Staubli VAL3: XHS3023L2.dtx

public frame fPartReal = {x=0.000, y=0.000, z=0.000, rx=0.000, ry=0.000, rz=0.000, fatherId=world[0]}
public jointRx jtPark = {j1=-10.678, j2=62.119, j3=50.568, j4=-4.773, j5=72.927, j6=-11.595}
public jointRx ptRoutingPath[1367]
  [0] = {j1=-10.951, j2=61.954, j3=48.631, j4=-3.846, j5=78.024, j6=-9.408}
  [1] = {j1=-10.927, j2=62.459, j3=48.172, j4=-3.903, j5=78.392, j6=-8.968}
  [2] = {j1=-10.905, j2=62.967, j3=47.706, j4=-3.960, j5=78.777, j6=-8.517}
  [3] = {j1=-10.884, j2=63.472, j3=47.245, j4=-4.014, j5=79.163, j6=-8.066}
  [4] = {j1=-10.866, j2=63.967, j3=46.802, j4=-4.064, j5=79.533, j6=-7.626}
  [5] = {j1=-10.851, j2=64.445, j3=46.388, j4=-4.105, j5=79.872, j6=-7.209}
  [6] = {j1=-10.848, j2=64.525, j3=46.320, j4=-4.112, j5=79.926, j6=-7.139}
  [7] = {j1=-10.829, j2=64.971, j3=45.959, j4=-4.174, j5=80.205, j6=-6.748}
  [8] = {j1=-10.797, j2=65.452, j3=45.616, j4=-4.291, j5=80.435, j6=-6.319}
  [9] = {j1=-10.755, j2=65.869, j3=45.388, j4=-4.456, j5=80.522, j6=-5.949}
  [10] = {j1=-10.719, j2=66.156, j3=45.303, j4=-4.610, j5=80.466, j6=-5.711}
  [11] = {j1=-10.683, j2=66.396, j3=45.302, j4=-4.767, j5=80.303, j6=-5.536}
  [12] = {j1=-10.648, j2=66.596, j3=45.373, j4=-4.931, j5=80.045, j6=-5.415}
  [13] = {j1=-10.612, j2=66.760, j3=45.504, j4=-5.105, j5=79.706, j6=-5.342}
  [14] = {j1=-10.575, j2=66.893, j3=45.686, j4=-5.292, j5=79.297, j6=-5.306}
  [15] = {j1=-10.535, j2=67.000, j3=45.908, j4=-5.496, j5=78.831, j6=-5.299}
  [16] = {j1=-10.534, j2=67.028, j3=45.859, j4=-5.501, j5=78.919, j6=-5.235}
  [17] = {j1=-10.574, j2=66.920, j3=45.638, j4=-5.295, j5=79.383, j6=-5.242}
  [18] = {j1=-10.612, j2=66.787, j3=45.457, j4=-5.107, j5=79.790, j6=-5.279}
  [19] = {j1=-10.648, j2=66.623, j3=45.325, j4=-4.932, j5=80.128, j6=-5.353}
  [20] = {j1=-10.683, j2=66.423, j3=45.255, j4=-4.767, j5=80.383, j6=-5.474}
  [21] = {j1=-10.719, j2=66.182, j3=45.257, j4=-4.608, j5=80.544, j6=-5.650}
  [22] = {j1=-10.756, j2=65.894, j3=45.344, j4=-4.452, j5=80.597, j6=-5.890}
  [23] = {j1=-10.798, j2=65.475, j3=45.576, j4=-4.285, j5=80.504, j6=-6.264}
  [24] = {j1=-10.831, j2=64.992, j3=45.924, j4=-4.167, j5=80.268, j6=-6.695}
  [25] = {j1=-10.850, j2=64.544, j3=46.288, j4=-4.104, j5=79.984, j6=-7.089}
  [26] = {j1=-10.853, j2=64.462, j3=46.358, j4=-4.097, j5=79.928, j6=-7.159}
  [27] = {j1=-10.868, j2=63.983, j3=46.774, j4=-4.055, j5=79.586, j6=-7.577}
  [28] = {j1=-10.887, j2=63.488, j3=47.217, j4=-4.005, j5=79.214, j6=-8.017}
  [29] = {j1=-10.908, j2=62.983, j3=47.678, j4=-3.950, j5=78.829, j6=-8.467}
  [30] = {j1=-10.930, j2=62.475, j3=48.144, j4=-3.893, j5=78.444, j6=-8.917}
  [31] = {j1=-10.953, j2=61.970, j3=48.602, j4=-3.836, j5=78.076, j6=-9.356}
  [32] = {j1=-10.977, j2=61.477, j3=49.042, j4=-3.779, j5=77.740, j6=-9.772}
  [33] = {j1=-10.999, j2=61.001, j3=49.449, j4=-3.727, j5=77.452, j6=-10.155}
  [34] = {j1=-11.016, j2=60.605, j3=49.771, j4=-3.691, j5=77.250, j6=-10.452}
  [35] = {j1=-11.028, j2=60.224, j3=50.065, j4=-3.672, j5=77.085, j6=-10.713}
  [36] = {j1=-11.036, j2=59.854, j3=50.341, j4=-3.667, j5=76.948, j6=-10.946}
  [37] = {j1=-11.039, j2=59.490, j3=50.605, j4=-3.676, j5=76.826, j6=-11.161}
  [38] = {j1=-11.039, j2=59.476, j3=50.615, j4=-3.676, j5=76.821, j6=-11.169}
  [39] = {j1=-11.040, j2=59.507, j3=50.561, j4=-3.671, j5=76.901, j6=-11.119}
  [40] = {j1=-11.040, j2=59.520, j3=50.552, j4=-3.671, j5=76.904, j6=-11.111}
  [41] = {j1=-11.037, j2=59.883, j3=50.289, j4=-3.662, j5=77.025, j6=-10.896}
  [42] = {j1=-11.029, j2=60.253, j3=50.015, j4=-3.666, j5=77.162, j6=-10.660}
  [43] = {j1=-11.018, j2=60.633, j3=49.721, j4=-3.684, j5=77.326, j6=-10.398}
  [44] = {j1=-11.001, j2=61.029, j3=49.400, j4=-3.719, j5=77.528, j6=-10.101}
  [45] = {j1=-10.979, j2=61.503, j3=48.995, j4=-3.772, j5=77.813, j6=-9.718}
  [46] = {j1=-10.955, j2=61.995, j3=48.559, j4=-3.827, j5=78.145, j6=-9.303}
  [47] = {j1=-10.932, j2=62.497, j3=48.105, j4=-3.885, j5=78.508, j6=-8.865}
  [48] = {j1=-10.910, j2=63.003, j3=47.644, j4=-3.941, j5=78.888, j6=-8.417}
  [49] = {j1=-10.889, j2=63.505, j3=47.187, j4=-3.996, j5=79.269, j6=-7.968}
  [50] = {j1=-10.871, j2=63.999, j3=46.747, j4=-4.045, j5=79.637, j6=-7.529}
  [51] = {j1=-10.855, j2=64.477, j3=46.332, j4=-4.088, j5=79.978, j6=-7.110}
  [52] = {j1=-10.853, j2=64.558, j3=46.264, j4=-4.095, j5=80.032, j6=-7.039}
  [53] = {j1=-10.833, j2=65.006, j3=45.900, j4=-4.158, j5=80.317, j6=-6.643}
  [54] = {j1=-10.800, j2=65.489, j3=45.550, j4=-4.278, j5=80.555, j6=-6.208}
  [55] = {j1=-10.758, j2=65.909, j3=45.318, j4=-4.446, j5=80.649, j6=-5.831}
  [56] = {j1=-10.720, j2=66.197, j3=45.232, j4=-4.603, j5=80.596, j6=-5.589}
  [57] = {j1=-10.684, j2=66.437, j3=45.231, j4=-4.763, j5=80.433, j6=-5.411}
  [58] = {j1=-10.649, j2=66.635, j3=45.304, j4=-4.930, j5=80.175, j6=-5.290}
  [59] = {j1=-10.612, j2=66.798, j3=45.438, j4=-5.105, j5=79.834, j6=-5.215}
  [60] = {j1=-10.574, j2=66.930, j3=45.622, j4=-5.294, j5=79.425, j6=-5.178}
  [61] = {j1=-10.534, j2=67.036, j3=45.845, j4=-5.501, j5=78.959, j6=-5.169}
  [62] = {j1=-10.533, j2=67.056, j3=45.811, j4=-5.504, j5=79.020, j6=-5.125}
  [63] = {j1=-10.574, j2=66.949, j3=45.589, j4=-5.297, j5=79.483, j6=-5.134}
  [64] = {j1=-10.612, j2=66.816, j3=45.406, j4=-5.107, j5=79.891, j6=-5.171}
  [65] = {j1=-10.649, j2=66.654, j3=45.273, j4=-4.930, j5=80.230, j6=-5.246}
  [66] = {j1=-10.685, j2=66.454, j3=45.201, j4=-4.763, j5=80.486, j6=-5.368}
  [67] = {j1=-10.721, j2=66.213, j3=45.203, j4=-4.601, j5=80.646, j6=-5.546}
  [68] = {j1=-10.759, j2=65.925, j3=45.292, j4=-4.443, j5=80.696, j6=-5.789}
  [69] = {j1=-10.802, j2=65.502, j3=45.527, j4=-4.273, j5=80.597, j6=-6.169}
  [70] = {j1=-10.835, j2=65.016, j3=45.881, j4=-4.152, j5=80.353, j6=-6.607}
  [71] = {j1=-10.854, j2=64.566, j3=46.249, j4=-4.089, j5=80.064, j6=-7.005}
  [72] = {j1=-10.857, j2=64.484, j3=46.319, j4=-4.081, j5=80.007, j6=-7.075}
  [73] = {j1=-10.873, j2=64.005, j3=46.736, j4=-4.038, j5=79.663, j6=-7.495}
  [74] = {j1=-10.891, j2=63.511, j3=47.177, j4=-3.988, j5=79.294, j6=-7.934}
  [75] = {j1=-10.912, j2=63.008, j3=47.634, j4=-3.934, j5=78.912, j6=-8.382}
  [76] = {j1=-10.934, j2=62.503, j3=48.095, j4=-3.876, j5=78.532, j6=-8.830}
  [77] = {j1=-10.958, j2=62.000, j3=48.550, j4=-3.819, j5=78.168, j6=-9.266}
  [78] = {j1=-10.981, j2=61.508, j3=48.986, j4=-3.763, j5=77.835, j6=-9.681}
  [79] = {j1=-11.003, j2=61.033, j3=49.393, j4=-3.711, j5=77.548, j6=-10.063}
  [80] = {j1=-11.020, j2=60.636, j3=49.717, j4=-3.676, j5=77.342, j6=-10.362}
  [81] = {j1=-11.032, j2=60.253, j3=50.015, j4=-3.657, j5=77.173, j6=-10.625}
  [82] = {j1=-11.039, j2=59.881, j3=50.293, j4=-3.653, j5=77.032, j6=-10.862}
  [83] = {j1=-11.043, j2=59.516, j3=50.559, j4=-3.662, j5=76.907, j6=-11.078}
  [84] = {j1=-11.043, j2=59.502, j3=50.570, j4=-3.662, j5=76.902, j6=-11.086}
  [85] = {j1=-11.044, j2=59.520, j3=50.538, j4=-3.659, j5=76.949, j6=-11.056}
  [86] = {j1=-11.044, j2=59.533, j3=50.529, j4=-3.659, j5=76.952, j6=-11.048}
  [87] = {j1=-11.040, j2=59.897, j3=50.265, j4=-3.649, j5=77.075, j6=-10.831}
  [88] = {j1=-11.033, j2=60.268, j3=49.988, j4=-3.653, j5=77.216, j6=-10.594}
  [89] = {j1=-11.021, j2=60.651, j3=49.690, j4=-3.671, j5=77.384, j6=-10.329}
  [90] = {j1=-11.005, j2=61.048, j3=49.368, j4=-3.706, j5=77.588, j6=-10.030}
  [91] = {j1=-10.982, j2=61.522, j3=48.963, j4=-3.758, j5=77.873, j6=-9.647}
  [92] = {j1=-10.959, j2=62.012, j3=48.530, j4=-3.813, j5=78.203, j6=-9.233}
  [93] = {j1=-10.936, j2=62.512, j3=48.079, j4=-3.870, j5=78.562, j6=-8.798}
  [94] = {j1=-10.914, j2=63.016, j3=47.622, j4=-3.927, j5=78.938, j6=-8.352}
  [95] = {j1=-10.893, j2=63.516, j3=47.168, j4=-3.982, j5=79.316, j6=-7.904}
  [96] = {j1=-10.875, j2=64.009, j3=46.729, j4=-4.031, j5=79.682, j6=-7.466}
  [97] = {j1=-10.859, j2=64.487, j3=46.315, j4=-4.074, j5=80.023, j6=-7.046}
  [98] = {j1=-10.856, j2=64.568, j3=46.247, j4=-4.082, j5=80.078, j6=-6.975}
  [99] = {j1=-10.837, j2=65.018, j3=45.879, j4=-4.145, j5=80.367, j6=-6.575}
  [100] = {j1=-10.803, j2=65.504, j3=45.525, j4=-4.267, j5=80.612, j6=-6.135}
  [101] = {j1=-10.760, j2=65.926, j3=45.289, j4=-4.437, j5=80.711, j6=-5.753}
  [102] = {j1=-10.722, j2=66.215, j3=45.201, j4=-4.597, j5=80.660, j6=-5.508}
  [103] = {j1=-10.686, j2=66.455, j3=45.201, j4=-4.759, j5=80.498, j6=-5.329}
  [104] = {j1=-10.649, j2=66.653, j3=45.275, j4=-4.927, j5=80.239, j6=-5.207}
  [105] = {j1=-10.613, j2=66.814, j3=45.411, j4=-5.104, j5=79.898, j6=-5.131}
  [106] = {j1=-10.575, j2=66.945, j3=45.596, j4=-5.294, j5=79.488, j6=-5.094}
  [107] = {j1=-10.534, j2=67.052, j3=45.819, j4=-5.502, j5=79.022, j6=-5.085}
  [108] = {j1=-10.533, j2=67.068, j3=45.789, j4=-5.505, j5=79.075, j6=-5.045}
  [109] = {j1=-10.574, j2=66.962, j3=45.567, j4=-5.296, j5=79.538, j6=-5.055}
  [110] = {j1=-10.613, j2=66.830, j3=45.383, j4=-5.105, j5=79.947, j6=-5.093}
  [111] = {j1=-10.649, j2=66.668, j3=45.249, j4=-4.927, j5=80.286, j6=-5.168}
  [112] = {j1=-10.686, j2=66.469, j3=45.176, j4=-4.758, j5=80.543, j6=-5.291}
  [113] = {j1=-10.723, j2=66.228, j3=45.178, j4=-4.595, j5=80.703, j6=-5.470}
  [114] = {j1=-10.761, j2=65.938, j3=45.268, j4=-4.434, j5=80.750, j6=-5.716}
  [115] = {j1=-10.804, j2=65.514, j3=45.507, j4=-4.262, j5=80.645, j6=-6.101}
  [116] = {j1=-10.838, j2=65.025, j3=45.866, j4=-4.140, j5=80.395, j6=-6.543}
  [117] = {j1=-10.858, j2=64.574, j3=46.237, j4=-4.075, j5=80.101, j6=-6.945}
  [118] = {j1=-10.861, j2=64.491, j3=46.307, j4=-4.068, j5=80.044, j6=-7.016}
  [119] = {j1=-10.876, j2=64.012, j3=46.724, j4=-4.024, j5=79.699, j6=-7.436}
  [120] = {j1=-10.895, j2=63.519, j3=47.164, j4=-3.974, j5=79.331, j6=-7.875}
  [121] = {j1=-10.916, j2=63.018, j3=47.618, j4=-3.920, j5=78.953, j6=-8.321}
  [122] = {j1=-10.938, j2=62.514, j3=48.076, j4=-3.863, j5=78.577, j6=-8.767}
  [123] = {j1=-10.961, j2=62.013, j3=48.527, j4=-3.805, j5=78.216, j6=-9.201}
  [124] = {j1=-10.984, j2=61.522, j3=48.962, j4=-3.750, j5=77.885, j6=-9.614}
  [125] = {j1=-11.007, j2=61.047, j3=49.368, j4=-3.698, j5=77.598, j6=-9.997}
  [126] = {j1=-11.023, j2=60.649, j3=49.694, j4=-3.663, j5=77.390, j6=-10.297}
  [127] = {j1=-11.035, j2=60.264, j3=49.995, j4=-3.645, j5=77.217, j6=-10.563}
  [128] = {j1=-11.043, j2=59.891, j3=50.276, j4=-3.641, j5=77.071, j6=-10.801}
  [129] = {j1=-11.046, j2=59.525, j3=50.544, j4=-3.650, j5=76.945, j6=-11.019}
  [130] = {j1=-11.046, j2=59.511, j3=50.554, j4=-3.650, j5=76.939, j6=-11.027}
  [131] = {j1=-11.047, j2=59.542, j3=50.500, j4=-3.645, j5=77.019, j6=-10.976}
  [132] = {j1=-11.047, j2=59.555, j3=50.492, j4=-3.644, j5=77.022, j6=-10.969}
  [133] = {j1=-11.044, j2=59.920, j3=50.225, j4=-3.635, j5=77.148, j6=-10.750}
  [134] = {j1=-11.037, j2=60.293, j3=49.944, j4=-3.638, j5=77.294, j6=-10.510}
  [135] = {j1=-11.025, j2=60.677, j3=49.643, j4=-3.656, j5=77.467, j6=-10.242}
  [136] = {j1=-11.009, j2=61.076, j3=49.319, j4=-3.691, j5=77.674, j6=-9.941}
  [137] = {j1=-10.986, j2=61.549, j3=48.915, j4=-3.742, j5=77.959, j6=-9.559}
  [138] = {j1=-10.963, j2=62.037, j3=48.485, j4=-3.797, j5=78.285, j6=-9.146}
  [139] = {j1=-10.940, j2=62.535, j3=48.039, j4=-3.854, j5=78.639, j6=-8.714}
  [140] = {j1=-10.918, j2=63.036, j3=47.586, j4=-3.910, j5=79.010, j6=-8.271}
  [141] = {j1=-10.898, j2=63.534, j3=47.137, j4=-3.965, j5=79.383, j6=-7.825}
  [142] = {j1=-10.879, j2=64.025, j3=46.701, j4=-4.015, j5=79.746, j6=-7.388}
  [143] = {j1=-10.863, j2=64.504, j3=46.286, j4=-4.058, j5=80.089, j6=-6.966}
  [144] = {j1=-10.861, j2=64.585, j3=46.218, j4=-4.066, j5=80.144, j6=-6.895}
  [145] = {j1=-10.841, j2=65.037, j3=45.846, j4=-4.130, j5=80.438, j6=-6.491}
  [146] = {j1=-10.807, j2=65.527, j3=45.486, j4=-4.254, j5=80.692, j6=-6.044}
  [147] = {j1=-10.763, j2=65.952, j3=45.245, j4=-4.427, j5=80.798, j6=-5.656}
  [148] = {j1=-10.724, j2=66.241, j3=45.156, j4=-4.589, j5=80.750, j6=-5.407}
  [149] = {j1=-10.687, j2=66.481, j3=45.156, j4=-4.754, j5=80.589, j6=-5.226}
  [150] = {j1=-10.650, j2=66.678, j3=45.231, j4=-4.924, j5=80.330, j6=-5.103}
  [151] = {j1=-10.613, j2=66.839, j3=45.369, j4=-5.103, j5=79.987, j6=-5.027}
  [152] = {j1=-10.575, j2=66.969, j3=45.556, j4=-5.295, j5=79.575, j6=-4.989}
  [153] = {j1=-10.534, j2=67.074, j3=45.780, j4=-5.504, j5=79.110, j6=-4.979}
  [154] = {j1=-10.532, j2=67.103, j3=45.730, j4=-5.509, j5=79.199, j6=-4.914}
  [155] = {j1=-10.574, j2=66.997, j3=45.507, j4=-5.298, j5=79.662, j6=-4.924}
  [156] = {j1=-10.613, j2=66.867, j3=45.320, j4=-5.105, j5=80.072, j6=-4.962}
  [157] = {j1=-10.650, j2=66.706, j3=45.183, j4=-4.925, j5=80.413, j6=-5.038}
  [158] = {j1=-10.687, j2=66.508, j3=45.109, j4=-4.753, j5=80.670, j6=-5.162}
  [159] = {j1=-10.724, j2=66.267, j3=45.110, j4=-4.587, j5=80.828, j6=-5.345}
  [160] = {j1=-10.763, j2=65.976, j3=45.202, j4=-4.423, j5=80.872, j6=-5.595}
  [161] = {j1=-10.808, j2=65.548, j3=45.448, j4=-4.248, j5=80.758, j6=-5.987}
  [162] = {j1=-10.843, j2=65.055, j3=45.814, j4=-4.122, j5=80.496, j6=-6.439}
  [163] = {j1=-10.863, j2=64.600, j3=46.191, j4=-4.057, j5=80.196, j6=-6.845}
  [164] = {j1=-10.866, j2=64.518, j3=46.262, j4=-4.049, j5=80.138, j6=-6.917}
  [165] = {j1=-10.882, j2=64.038, j3=46.679, j4=-4.005, j5=79.792, j6=-7.339}
  [166] = {j1=-10.900, j2=63.547, j3=47.116, j4=-3.955, j5=79.427, j6=-7.776}
  [167] = {j1=-10.921, j2=63.048, j3=47.564, j4=-3.900, j5=79.054, j6=-8.220}
  [168] = {j1=-10.943, j2=62.548, j3=48.016, j4=-3.843, j5=78.685, j6=-8.661}
  [169] = {j1=-10.966, j2=62.051, j3=48.461, j4=-3.786, j5=78.331, j6=-9.092}
  [170] = {j1=-10.989, j2=61.563, j3=48.891, j4=-3.731, j5=78.005, j6=-9.503}
  [171] = {j1=-11.011, j2=61.088, j3=49.297, j4=-3.680, j5=77.717, j6=-9.885}
  [172] = {j1=-11.028, j2=60.688, j3=49.625, j4=-3.645, j5=77.506, j6=-10.187}
  [173] = {j1=-11.040, j2=60.301, j3=49.930, j4=-3.627, j5=77.327, j6=-10.457}
  [174] = {j1=-11.047, j2=59.925, j3=50.216, j4=-3.624, j5=77.175, j6=-10.699}
  [175] = {j1=-11.050, j2=59.558, j3=50.487, j4=-3.633, j5=77.045, j6=-10.919}
  [176] = {j1=-11.051, j2=59.544, j3=50.497, j4=-3.634, j5=77.039, j6=-10.927}
  [177] = {j1=-11.052, j2=59.575, j3=50.442, j4=-3.629, j5=77.120, j6=-10.876}
  [178] = {j1=-11.052, j2=59.588, j3=50.434, j4=-3.628, j5=77.123, j6=-10.868}
  [179] = {j1=-11.048, j2=59.954, j3=50.164, j4=-3.618, j5=77.253, j6=-10.647}
  [180] = {j1=-11.041, j2=60.330, j3=49.879, j4=-3.621, j5=77.405, j6=-10.403}
  [181] = {j1=-11.030, j2=60.717, j3=49.574, j4=-3.638, j5=77.583, j6=-10.132}
  [182] = {j1=-11.013, j2=61.116, j3=49.247, j4=-3.672, j5=77.794, j6=-9.829}
  [183] = {j1=-10.991, j2=61.589, j3=48.845, j4=-3.723, j5=78.077, j6=-9.447}
  [184] = {j1=-10.968, j2=62.075, j3=48.420, j4=-3.778, j5=78.399, j6=-9.037}
  [185] = {j1=-10.946, j2=62.569, j3=47.980, j4=-3.834, j5=78.746, j6=-8.609}
  [186] = {j1=-10.924, j2=63.066, j3=47.534, j4=-3.891, j5=79.109, j6=-8.169}
  [187] = {j1=-10.903, j2=63.561, j3=47.091, j4=-3.945, j5=79.476, j6=-7.727}
  [188] = {j1=-10.884, j2=64.050, j3=46.658, j4=-3.995, j5=79.836, j6=-7.291}
  [189] = {j1=-10.869, j2=64.529, j3=46.243, j4=-4.039, j5=80.179, j6=-6.868}
  [190] = {j1=-10.866, j2=64.610, j3=46.174, j4=-4.046, j5=80.235, j6=-6.796}
  [191] = {j1=-10.845, j2=65.065, j3=45.798, j4=-4.112, j5=80.536, j6=-6.387}
  [192] = {j1=-10.810, j2=65.559, j3=45.430, j4=-4.239, j5=80.801, j6=-5.931}
  [193] = {j1=-10.765, j2=65.988, j3=45.183, j4=-4.416, j5=80.917, j6=-5.535}
  [194] = {j1=-10.726, j2=66.278, j3=45.091, j4=-4.581, j5=80.873, j6=-5.282}
  [195] = {j1=-10.688, j2=66.518, j3=45.092, j4=-4.749, j5=80.712, j6=-5.098}
  [196] = {j1=-10.651, j2=66.714, j3=45.169, j4=-4.921, j5=80.452, j6=-4.973}
  [197] = {j1=-10.613, j2=66.874, j3=45.309, j4=-5.103, j5=80.108, j6=-4.897}
  [198] = {j1=-10.574, j2=67.002, j3=45.498, j4=-5.297, j5=79.695, j6=-4.859}
  [199] = {j1=-10.533, j2=67.107, j3=45.724, j4=-5.508, j5=79.229, j6=-4.847}
  [200] = {j1=-10.532, j2=67.135, j3=45.675, j4=-5.513, j5=79.318, j6=-4.782}
  [201] = {j1=-10.574, j2=67.030, j3=45.450, j4=-5.300, j5=79.781, j6=-4.794}
  [202] = {j1=-10.613, j2=66.901, j3=45.261, j4=-5.105, j5=80.192, j6=-4.832}
  [203] = {j1=-10.651, j2=66.741, j3=45.122, j4=-4.922, j5=80.534, j6=-4.909}
  [204] = {j1=-10.688, j2=66.545, j3=45.045, j4=-4.748, j5=80.792, j6=-5.034}
  [205] = {j1=-10.726, j2=66.304, j3=45.047, j4=-4.579, j5=80.949, j6=-5.219}
  [206] = {j1=-10.766, j2=66.011, j3=45.142, j4=-4.412, j5=80.988, j6=-5.475}
  [207] = {j1=-10.812, j2=65.579, j3=45.394, j4=-4.232, j5=80.864, j6=-5.876}
  [208] = {j1=-10.848, j2=65.082, j3=45.768, j4=-4.104, j5=80.592, j6=-6.336}
  [209] = {j1=-10.868, j2=64.624, j3=46.150, j4=-4.037, j5=80.285, j6=-6.748}
  [210] = {j1=-10.871, j2=64.541, j3=46.221, j4=-4.029, j5=80.225, j6=-6.820}
  [211] = {j1=-10.887, j2=64.061, j3=46.639, j4=-3.985, j5=79.878, j6=-7.243}
  [212] = {j1=-10.906, j2=63.572, j3=47.072, j4=-3.935, j5=79.517, j6=-7.679}
  [213] = {j1=-10.926, j2=63.077, j3=47.515, j4=-3.880, j5=79.150, j6=-8.119}
  [214] = {j1=-10.948, j2=62.580, j3=47.959, j4=-3.823, j5=78.789, j6=-8.556}
  [215] = {j1=-10.971, j2=62.087, j3=48.398, j4=-3.767, j5=78.442, j6=-8.982}
  [216] = {j1=-10.994, j2=61.601, j3=48.824, j4=-3.712, j5=78.121, j6=-9.390}
  [217] = {j1=-11.016, j2=61.128, j3=49.227, j4=-3.661, j5=77.834, j6=-9.773}
  [218] = {j1=-11.033, j2=60.726, j3=49.558, j4=-3.627, j5=77.619, j6=-10.077}
  [219] = {j1=-11.044, j2=60.337, j3=49.867, j4=-3.609, j5=77.435, j6=-10.349}
  [220] = {j1=-11.052, j2=59.958, j3=50.158, j4=-3.606, j5=77.277, j6=-10.595}
  [221] = {j1=-11.055, j2=59.589, j3=50.431, j4=-3.616, j5=77.142, j6=-10.818}
  [222] = {j1=-11.055, j2=59.575, j3=50.442, j4=-3.617, j5=77.136, j6=-10.825}
  [223] = {j1=-11.056, j2=59.607, j3=50.386, j4=-3.612, j5=77.219, j6=-10.774}
  [224] = {j1=-11.056, j2=59.620, j3=50.378, j4=-3.611, j5=77.222, j6=-10.766}
  [225] = {j1=-11.053, j2=59.988, j3=50.105, j4=-3.600, j5=77.356, j6=-10.542}
  [226] = {j1=-11.046, j2=60.366, j3=49.815, j4=-3.603, j5=77.513, j6=-10.295}
  [227] = {j1=-11.034, j2=60.755, j3=49.507, j4=-3.620, j5=77.697, j6=-10.020}
  [228] = {j1=-11.018, j2=61.156, j3=49.178, j4=-3.653, j5=77.910, j6=-9.716}
  [229] = {j1=-10.996, j2=61.627, j3=48.778, j4=-3.704, j5=78.193, j6=-9.334}
  [230] = {j1=-10.973, j2=62.110, j3=48.358, j4=-3.758, j5=78.508, j6=-8.927}
  [231] = {j1=-10.951, j2=62.600, j3=47.925, j4=-3.814, j5=78.848, j6=-8.503}
  [232] = {j1=-10.929, j2=63.093, j3=47.487, j4=-3.871, j5=79.203, j6=-8.068}
  [233] = {j1=-10.908, j2=63.585, j3=47.050, j4=-3.925, j5=79.563, j6=-7.630}
  [234] = {j1=-10.890, j2=64.072, j3=46.621, j4=-3.975, j5=79.919, j6=-7.196}
  [235] = {j1=-10.874, j2=64.550, j3=46.205, j4=-4.019, j5=80.264, j6=-6.772}
  [236] = {j1=-10.871, j2=64.632, j3=46.136, j4=-4.027, j5=80.320, j6=-6.699}
  [237] = {j1=-10.850, j2=65.090, j3=45.755, j4=-4.094, j5=80.628, j6=-6.284}
  [238] = {j1=-10.815, j2=65.588, j3=45.379, j4=-4.223, j5=80.903, j6=-5.820}
  [239] = {j1=-10.768, j2=66.021, j3=45.125, j4=-4.404, j5=81.029, j6=-5.415}
  [240] = {j1=-10.728, j2=66.313, j3=45.031, j4=-4.573, j5=80.989, j6=-5.157}
  [241] = {j1=-10.689, j2=66.553, j3=45.031, j4=-4.743, j5=80.831, j6=-4.970}
  [242] = {j1=-10.652, j2=66.748, j3=45.110, j4=-4.918, j5=80.570, j6=-4.844}
  [243] = {j1=-10.614, j2=66.906, j3=45.253, j4=-5.102, j5=80.224, j6=-4.767}
  [244] = {j1=-10.574, j2=67.034, j3=45.444, j4=-5.298, j5=79.810, j6=-4.728}
  [245] = {j1=-10.532, j2=67.138, j3=45.672, j4=-5.511, j5=79.344, j6=-4.715}
  [246] = {j1=-10.531, j2=67.166, j3=45.622, j4=-5.516, j5=79.432, j6=-4.650}
  [247] = {j1=-10.573, j2=67.062, j3=45.396, j4=-5.302, j5=79.896, j6=-4.663}
  [248] = {j1=-10.613, j2=66.934, j3=45.205, j4=-5.104, j5=80.308, j6=-4.703}
  [249] = {j1=-10.651, j2=66.775, j3=45.064, j4=-4.919, j5=80.651, j6=-4.780}
  [250] = {j1=-10.690, j2=66.579, j3=44.986, j4=-4.742, j5=80.909, j6=-4.907}
  [251] = {j1=-10.729, j2=66.338, j3=44.988, j4=-4.570, j5=81.064, j6=-5.095}
  [252] = {j1=-10.769, j2=66.044, j3=45.085, j4=-4.400, j5=81.099, j6=-5.355}
  [253] = {j1=-10.816, j2=65.608, j3=45.345, j4=-4.216, j5=80.965, j6=-5.765}
  [254] = {j1=-10.853, j2=65.105, j3=45.727, j4=-4.085, j5=80.681, j6=-6.233}
  [255] = {j1=-10.874, j2=64.645, j3=46.114, j4=-4.017, j5=80.367, j6=-6.651}
  [256] = {j1=-10.877, j2=64.562, j3=46.186, j4=-4.009, j5=80.306, j6=-6.724}
  [257] = {j1=-10.893, j2=64.082, j3=46.604, j4=-3.965, j5=79.958, j6=-7.148}
  [258] = {j1=-10.911, j2=63.594, j3=47.033, j4=-3.914, j5=79.601, j6=-7.582}
  [259] = {j1=-10.932, j2=63.103, j3=47.470, j4=-3.860, j5=79.241, j6=-8.018}
  [260] = {j1=-10.954, j2=62.610, j3=47.907, j4=-3.803, j5=78.888, j6=-8.450}
  [261] = {j1=-10.976, j2=62.121, j3=48.339, j4=-3.747, j5=78.549, j6=-8.872}
  [262] = {j1=-10.999, j2=61.638, j3=48.759, j4=-3.693, j5=78.233, j6=-9.277}
  [263] = {j1=-11.021, j2=61.166, j3=49.161, j4=-3.642, j5=77.948, j6=-9.659}
  [264] = {j1=-11.037, j2=60.763, j3=49.493, j4=-3.608, j5=77.730, j6=-9.964}
  [265] = {j1=-11.049, j2=60.372, j3=49.806, j4=-3.590, j5=77.541, j6=-10.240}
  [266] = {j1=-11.056, j2=59.991, j3=50.101, j4=-3.588, j5=77.377, j6=-10.490}
  [267] = {j1=-11.059, j2=59.620, j3=50.378, j4=-3.599, j5=77.238, j6=-10.715}
  [268] = {j1=-11.060, j2=59.606, j3=50.389, j4=-3.599, j5=77.231, j6=-10.722}
  [269] = {j1=-11.061, j2=59.638, j3=50.332, j4=-3.594, j5=77.315, j6=-10.670}
  [270] = {j1=-11.061, j2=59.651, j3=50.323, j4=-3.593, j5=77.318, j6=-10.662}
  [271] = {j1=-11.058, j2=60.021, j3=50.048, j4=-3.582, j5=77.456, j6=-10.436}
  [272] = {j1=-11.051, j2=60.401, j3=49.754, j4=-3.584, j5=77.619, j6=-10.185}
  [273] = {j1=-11.039, j2=60.792, j3=49.442, j4=-3.600, j5=77.808, j6=-9.908}
  [274] = {j1=-11.023, j2=61.194, j3=49.111, j4=-3.634, j5=78.024, j6=-9.601}
  [275] = {j1=-11.001, j2=61.664, j3=48.714, j4=-3.685, j5=78.304, j6=-9.220}
  [276] = {j1=-10.978, j2=62.143, j3=48.299, j4=-3.739, j5=78.614, j6=-8.817}
  [277] = {j1=-10.956, j2=62.629, j3=47.874, j4=-3.794, j5=78.945, j6=-8.398}
  [278] = {j1=-10.934, j2=63.118, j3=47.444, j4=-3.850, j5=79.291, j6=-7.968}
  [279] = {j1=-10.914, j2=63.606, j3=47.013, j4=-3.904, j5=79.644, j6=-7.533}
  [280] = {j1=-10.896, j2=64.091, j3=46.588, j4=-3.955, j5=79.996, j6=-7.101}
  [281] = {j1=-10.879, j2=64.569, j3=46.173, j4=-3.999, j5=80.341, j6=-6.676}
  [282] = {j1=-10.877, j2=64.651, j3=46.103, j4=-4.006, j5=80.399, j6=-6.603}
  [283] = {j1=-10.856, j2=65.112, j3=45.717, j4=-4.074, j5=80.713, j6=-6.183}
  [284] = {j1=-10.819, j2=65.615, j3=45.332, j4=-4.206, j5=81.000, j6=-5.709}
  [285] = {j1=-10.772, j2=66.052, j3=45.072, j4=-4.391, j5=81.136, j6=-5.295}
  [286] = {j1=-10.730, j2=66.346, j3=44.975, j4=-4.564, j5=81.101, j6=-5.032}
  [287] = {j1=-10.691, j2=66.586, j3=44.975, j4=-4.737, j5=80.943, j6=-4.843}
  [288] = {j1=-10.653, j2=66.780, j3=45.056, j4=-4.915, j5=80.682, j6=-4.715}
  [289] = {j1=-10.614, j2=66.937, j3=45.200, j4=-5.101, j5=80.335, j6=-4.637}
  [290] = {j1=-10.574, j2=67.063, j3=45.394, j4=-5.299, j5=79.920, j6=-4.597}
  [291] = {j1=-10.532, j2=67.166, j3=45.623, j4=-5.514, j5=79.453, j6=-4.584}
  [292] = {j1=-10.531, j2=67.194, j3=45.574, j4=-5.518, j5=79.542, j6=-4.519}
  [293] = {j1=-10.573, j2=67.091, j3=45.346, j4=-5.303, j5=80.005, j6=-4.533}
  [294] = {j1=-10.613, j2=66.964, j3=45.153, j4=-5.103, j5=80.418, j6=-4.573}
  [295] = {j1=-10.652, j2=66.807, j3=45.010, j4=-4.916, j5=80.763, j6=-4.651}
  [296] = {j1=-10.691, j2=66.611, j3=44.931, j4=-4.736, j5=81.021, j6=-4.780}
  [297] = {j1=-10.731, j2=66.370, j3=44.933, j4=-4.561, j5=81.174, j6=-4.971}
  [298] = {j1=-10.773, j2=66.074, j3=45.033, j4=-4.387, j5=81.203, j6=-5.236}
  [299] = {j1=-10.821, j2=65.634, j3=45.301, j4=-4.199, j5=81.059, j6=-5.654}
  [300] = {j1=-10.858, j2=65.126, j3=45.692, j4=-4.065, j5=80.764, j6=-6.132}
  [301] = {j1=-10.879, j2=64.663, j3=46.083, j4=-3.996, j5=80.442, j6=-6.555}
  [302] = {j1=-10.882, j2=64.579, j3=46.156, j4=-3.989, j5=80.381, j6=-6.628}
  [303] = {j1=-10.898, j2=64.099, j3=46.573, j4=-3.944, j5=80.032, j6=-7.054}
  [304] = {j1=-10.917, j2=63.614, j3=46.999, j4=-3.894, j5=79.679, j6=-7.485}
  [305] = {j1=-10.937, j2=63.126, j3=47.429, j4=-3.839, j5=79.326, j6=-7.917}
  [306] = {j1=-10.959, j2=62.638, j3=47.859, j4=-3.783, j5=78.982, j6=-8.345}
  [307] = {j1=-10.981, j2=62.153, j3=48.283, j4=-3.727, j5=78.651, j6=-8.762}
  [308] = {j1=-11.004, j2=61.673, j3=48.697, j4=-3.673, j5=78.341, j6=-9.163}
  [309] = {j1=-11.026, j2=61.202, j3=49.097, j4=-3.622, j5=78.059, j6=-9.544}
  [310] = {j1=-11.042, j2=60.799, j3=49.430, j4=-3.588, j5=77.839, j6=-9.851}
  [311] = {j1=-11.054, j2=60.405, j3=49.747, j4=-3.571, j5=77.644, j6=-10.130}
  [312] = {j1=-11.061, j2=60.022, j3=50.047, j4=-3.569, j5=77.474, j6=-10.383}
  [313] = {j1=-11.064, j2=59.649, j3=50.327, j4=-3.580, j5=77.330, j6=-10.610}
  [314] = {j1=-11.064, j2=59.635, j3=50.338, j4=-3.581, j5=77.324, j6=-10.618}
  [315] = {j1=-11.065, j2=59.668, j3=50.280, j4=-3.576, j5=77.408, j6=-10.565}
  [316] = {j1=-11.065, j2=59.680, j3=50.272, j4=-3.575, j5=77.411, j6=-10.557}
  [317] = {j1=-11.062, j2=60.052, j3=49.993, j4=-3.563, j5=77.554, j6=-10.328}
  [318] = {j1=-11.055, j2=60.435, j3=49.695, j4=-3.564, j5=77.723, j6=-10.074}
  [319] = {j1=-11.044, j2=60.828, j3=49.379, j4=-3.581, j5=77.917, j6=-9.794}
  [320] = {j1=-11.028, j2=61.230, j3=49.048, j4=-3.614, j5=78.134, j6=-9.486}
  [321] = {j1=-11.006, j2=61.698, j3=48.653, j4=-3.665, j5=78.412, j6=-9.106}
  [322] = {j1=-10.983, j2=62.175, j3=48.245, j4=-3.718, j5=78.715, j6=-8.706}
  [323] = {j1=-10.961, j2=62.656, j3=47.827, j4=-3.774, j5=79.037, j6=-8.292}
  [324] = {j1=-10.940, j2=63.140, j3=47.405, j4=-3.830, j5=79.374, j6=-7.867}
  [325] = {j1=-10.920, j2=63.625, j3=46.981, j4=-3.884, j5=79.719, j6=-7.437}
  [326] = {j1=-10.901, j2=64.107, j3=46.560, j4=-3.933, j5=80.067, j6=-7.007}
  [327] = {j1=-10.885, j2=64.585, j3=46.146, j4=-3.978, j5=80.413, j6=-6.581}
  [328] = {j1=-10.883, j2=64.667, j3=46.075, j4=-3.985, j5=80.471, j6=-6.507}
  [329] = {j1=-10.861, j2=65.131, j3=45.684, j4=-4.054, j5=80.792, j6=-6.082}
  [330] = {j1=-10.824, j2=65.639, j3=45.291, j4=-4.188, j5=81.090, j6=-5.600}
  [331] = {j1=-10.775, j2=66.080, j3=45.023, j4=-4.378, j5=81.236, j6=-5.177}
  [332] = {j1=-10.733, j2=66.375, j3=44.924, j4=-4.554, j5=81.206, j6=-4.909}
  [333] = {j1=-10.693, j2=66.616, j3=44.924, j4=-4.731, j5=81.050, j6=-4.716}
  [334] = {j1=-10.654, j2=66.810, j3=45.005, j4=-4.911, j5=80.789, j6=-4.586}
  [335] = {j1=-10.615, j2=66.965, j3=45.152, j4=-5.100, j5=80.441, j6=-4.507}
  [336] = {j1=-10.574, j2=67.091, j3=45.348, j4=-5.300, j5=80.025, j6=-4.467}
  [337] = {j1=-10.532, j2=67.193, j3=45.578, j4=-5.516, j5=79.558, j6=-4.453}
  [338] = {j1=-10.531, j2=67.221, j3=45.530, j4=-5.521, j5=79.646, j6=-4.388}
  [339] = {j1=-10.573, j2=67.118, j3=45.300, j4=-5.303, j5=80.110, j6=-4.403}
  [340] = {j1=-10.614, j2=66.992, j3=45.105, j4=-5.102, j5=80.523, j6=-4.443}
  [341] = {j1=-10.653, j2=66.836, j3=44.960, j4=-4.912, j5=80.868, j6=-4.522}
  [342] = {j1=-10.693, j2=66.641, j3=44.880, j4=-4.730, j5=81.126, j6=-4.653}
  [343] = {j1=-10.733, j2=66.399, j3=44.884, j4=-4.551, j5=81.277, j6=-4.847}
  [344] = {j1=-10.776, j2=66.101, j3=44.987, j4=-4.373, j5=81.301, j6=-5.118}
  [345] = {j1=-10.825, j2=65.656, j3=45.261, j4=-4.181, j5=81.147, j6=-5.545}
  [346] = {j1=-10.863, j2=65.144, j3=45.661, j4=-4.045, j5=80.840, j6=-6.032}
  [347] = {j1=-10.885, j2=64.678, j3=46.058, j4=-3.975, j5=80.511, j6=-6.459}
  [348] = {j1=-10.888, j2=64.594, j3=46.131, j4=-3.967, j5=80.450, j6=-6.533}
  [349] = {j1=-10.904, j2=64.114, j3=46.548, j4=-3.923, j5=80.100, j6=-6.959}
  [350] = {j1=-10.923, j2=63.631, j3=46.970, j4=-3.873, j5=79.751, j6=-7.389}
  [351] = {j1=-10.943, j2=63.147, j3=47.393, j4=-3.819, j5=79.406, j6=-7.817}
  [352] = {j1=-10.964, j2=62.664, j3=47.815, j4=-3.763, j5=79.070, j6=-8.239}
  [353] = {j1=-10.987, j2=62.183, j3=48.231, j4=-3.707, j5=78.749, j6=-8.651}
  [354] = {j1=-11.009, j2=61.707, j3=48.639, j4=-3.653, j5=78.445, j6=-9.049}
  [355] = {j1=-11.031, j2=61.237, j3=49.036, j4=-3.602, j5=78.166, j6=-9.428}
  [356] = {j1=-11.047, j2=60.833, j3=49.370, j4=-3.568, j5=77.943, j6=-9.736}
  [357] = {j1=-11.059, j2=60.437, j3=49.691, j4=-3.551, j5=77.744, j6=-10.019}
  [358] = {j1=-11.066, j2=60.051, j3=49.995, j4=-3.549, j5=77.569, j6=-10.274}
  [359] = {j1=-11.069, j2=59.677, j3=50.279, j4=-3.562, j5=77.419, j6=-10.505}
  [360] = {j1=-11.069, j2=59.662, j3=50.290, j4=-3.562, j5=77.413, j6=-10.513}
  [361] = {j1=-11.070, j2=59.696, j3=50.231, j4=-3.557, j5=77.498, j6=-10.459}
  [362] = {j1=-11.070, j2=59.708, j3=50.223, j4=-3.556, j5=77.501, j6=-10.451}
  [363] = {j1=-11.068, j2=60.082, j3=49.940, j4=-3.543, j5=77.649, j6=-10.219}
  [364] = {j1=-11.061, j2=60.467, j3=49.638, j4=-3.544, j5=77.823, j6=-9.962}
  [365] = {j1=-11.049, j2=60.862, j3=49.319, j4=-3.560, j5=78.021, j6=-9.678}
  [366] = {j1=-11.033, j2=61.264, j3=48.987, j4=-3.594, j5=78.241, j6=-9.369}
  [367] = {j1=-11.011, j2=61.731, j3=48.596, j4=-3.644, j5=78.515, j6=-8.991}
  [368] = {j1=-10.989, j2=62.204, j3=48.194, j4=-3.698, j5=78.811, j6=-8.595}
  [369] = {j1=-10.967, j2=62.681, j3=47.785, j4=-3.753, j5=79.124, j6=-8.185}
  [370] = {j1=-10.945, j2=63.160, j3=47.371, j4=-3.809, j5=79.451, j6=-7.766}
  [371] = {j1=-10.925, j2=63.640, j3=46.954, j4=-3.862, j5=79.789, j6=-7.340}
  [372] = {j1=-10.907, j2=64.120, j3=46.538, j4=-3.912, j5=80.132, j6=-6.913}
  [373] = {j1=-10.891, j2=64.598, j3=46.123, j4=-3.956, j5=80.478, j6=-6.486}
  [374] = {j1=-10.888, j2=64.681, j3=46.053, j4=-3.963, j5=80.536, j6=-6.412}
  [375] = {j1=-10.867, j2=65.147, j3=45.657, j4=-4.033, j5=80.865, j6=-5.982}
  [376] = {j1=-10.828, j2=65.660, j3=45.256, j4=-4.170, j5=81.174, j6=-5.491}
  [377] = {j1=-10.778, j2=66.105, j3=44.980, j4=-4.364, j5=81.330, j6=-5.059}
  [378] = {j1=-10.735, j2=66.402, j3=44.878, j4=-4.544, j5=81.304, j6=-4.785}
  [379] = {j1=-10.694, j2=66.643, j3=44.877, j4=-4.723, j5=81.151, j6=-4.589}
  [380] = {j1=-10.655, j2=66.836, j3=44.959, j4=-4.907, j5=80.890, j6=-4.458}
  [381] = {j1=-10.615, j2=66.991, j3=45.108, j4=-5.098, j5=80.541, j6=-4.378}
  [382] = {j1=-10.575, j2=67.115, j3=45.306, j4=-5.300, j5=80.124, j6=-4.337}
  [383] = {j1=-10.532, j2=67.217, j3=45.538, j4=-5.518, j5=79.656, j6=-4.321}
  [384] = {j1=-10.531, j2=67.245, j3=45.489, j4=-5.522, j5=79.744, j6=-4.257}
  [385] = {j1=-10.574, j2=67.143, j3=45.258, j4=-5.303, j5=80.208, j6=-4.272}
  [386] = {j1=-10.615, j2=67.018, j3=45.062, j4=-5.100, j5=80.623, j6=-4.314}
  [387] = {j1=-10.654, j2=66.862, j3=44.915, j4=-4.907, j5=80.968, j6=-4.394}
  [388] = {j1=-10.695, j2=66.667, j3=44.835, j4=-4.722, j5=81.225, j6=-4.526}
  [389] = {j1=-10.736, j2=66.425, j3=44.839, j4=-4.541, j5=81.374, j6=-4.724}
  [390] = {j1=-10.780, j2=66.125, j3=44.945, j4=-4.358, j5=81.393, j6=-5.000}
  [391] = {j1=-10.830, j2=65.676, j3=45.228, j4=-4.162, j5=81.228, j6=-5.437}
  [392] = {j1=-10.869, j2=65.159, j3=45.636, j4=-4.023, j5=80.910, j6=-5.932}
  [393] = {j1=-10.891, j2=64.690, j3=46.037, j4=-3.953, j5=80.574, j6=-6.365}
  [394] = {j1=-10.894, j2=64.606, j3=46.111, j4=-3.945, j5=80.512, j6=-6.439}
  [395] = {j1=-10.910, j2=64.126, j3=46.528, j4=-3.901, j5=80.162, j6=-6.866}
  [396] = {j1=-10.929, j2=63.645, j3=46.946, j4=-3.851, j5=79.817, j6=-7.292}
  [397] = {j1=-10.949, j2=63.165, j3=47.362, j4=-3.797, j5=79.480, j6=-7.715}
  [398] = {j1=-10.970, j2=62.686, j3=47.775, j4=-3.742, j5=79.154, j6=-8.132}
  [399] = {j1=-10.992, j2=62.210, j3=48.183, j4=-3.686, j5=78.841, j6=-8.539}
  [400] = {j1=-11.014, j2=61.738, j3=48.585, j4=-3.632, j5=78.545, j6=-8.933}
  [401] = {j1=-11.036, j2=61.270, j3=48.978, j4=-3.581, j5=78.269, j6=-9.311}
  [402] = {j1=-11.053, j2=60.865, j3=49.314, j4=-3.547, j5=78.045, j6=-9.621}
  [403] = {j1=-11.064, j2=60.468, j3=49.638, j4=-3.530, j5=77.841, j6=-9.905}
  [404] = {j1=-11.071, j2=60.080, j3=49.945, j4=-3.529, j5=77.660, j6=-10.165}
  [405] = {j1=-11.074, j2=59.703, j3=50.233, j4=-3.542, j5=77.505, j6=-10.398}
  [406] = {j1=-11.074, j2=59.688, j3=50.245, j4=-3.542, j5=77.498, j6=-10.406}
  [407] = {j1=-11.075, j2=59.722, j3=50.185, j4=-3.537, j5=77.585, j6=-10.352}
  [408] = {j1=-11.075, j2=59.735, j3=50.177, j4=-3.536, j5=77.588, j6=-10.344}
  [409] = {j1=-11.073, j2=60.111, j3=49.891, j4=-3.523, j5=77.741, j6=-10.109}
  [410] = {j1=-11.066, j2=60.498, j3=49.584, j4=-3.523, j5=77.920, j6=-9.848}
  [411] = {j1=-11.054, j2=60.894, j3=49.263, j4=-3.539, j5=78.122, j6=-9.562}
  [412] = {j1=-11.038, j2=61.297, j3=48.930, j4=-3.573, j5=78.343, j6=-9.251}
  [413] = {j1=-11.016, j2=61.762, j3=48.542, j4=-3.624, j5=78.613, j6=-8.875}
  [414] = {j1=-10.994, j2=62.231, j3=48.147, j4=-3.677, j5=78.902, j6=-8.483}
  [415] = {j1=-10.972, j2=62.703, j3=47.747, j4=-3.733, j5=79.206, j6=-8.079}
  [416] = {j1=-10.951, j2=63.177, j3=47.341, j4=-3.788, j5=79.523, j6=-7.665}
  [417] = {j1=-10.931, j2=63.653, j3=46.932, j4=-3.841, j5=79.852, j6=-7.244}
  [418] = {j1=-10.913, j2=64.131, j3=46.520, j4=-3.890, j5=80.191, j6=-6.819}
  [419] = {j1=-10.897, j2=64.609, j3=46.106, j4=-3.933, j5=80.536, j6=-6.392}
  [420] = {j1=-10.895, j2=64.691, j3=46.036, j4=-3.941, j5=80.595, j6=-6.317}
  [421] = {j1=-10.872, j2=65.160, j3=45.635, j4=-4.011, j5=80.930, j6=-5.882}
  [422] = {j1=-10.833, j2=65.678, j3=45.226, j4=-4.151, j5=81.250, j6=-5.383}
  [423] = {j1=-10.782, j2=66.127, j3=44.943, j4=-4.349, j5=81.417, j6=-4.942}
  [424] = {j1=-10.738, j2=66.426, j3=44.837, j4=-4.533, j5=81.396, j6=-4.662}
  [425] = {j1=-10.696, j2=66.667, j3=44.835, j4=-4.716, j5=81.245, j6=-4.463}
  [426] = {j1=-10.656, j2=66.861, j3=44.918, j4=-4.902, j5=80.985, j6=-4.329}
  [427] = {j1=-10.616, j2=67.014, j3=45.068, j4=-5.095, j5=80.635, j6=-4.248}
  [428] = {j1=-10.575, j2=67.138, j3=45.268, j4=-5.299, j5=80.217, j6=-4.206}
  [429] = {j1=-10.532, j2=67.238, j3=45.502, j4=-5.519, j5=79.749, j6=-4.190}
  [430] = {j1=-10.531, j2=67.266, j3=45.453, j4=-5.523, j5=79.836, j6=-4.126}
  [431] = {j1=-10.574, j2=67.165, j3=45.221, j4=-5.303, j5=80.300, j6=-4.142}
  [432] = {j1=-10.615, j2=67.040, j3=45.023, j4=-5.097, j5=80.716, j6=-4.184}
  [433] = {j1=-10.656, j2=66.885, j3=44.875, j4=-4.902, j5=81.062, j6=-4.266}
  [434] = {j1=-10.697, j2=66.691, j3=44.794, j4=-4.714, j5=81.318, j6=-4.400}
  [435] = {j1=-10.739, j2=66.448, j3=44.800, j4=-4.529, j5=81.464, j6=-4.601}
  [436] = {j1=-10.784, j2=66.146, j3=44.910, j4=-4.343, j5=81.478, j6=-4.883}
  [437] = {j1=-10.835, j2=65.693, j3=45.199, j4=-4.142, j5=81.303, j6=-5.329}
  [438] = {j1=-10.875, j2=65.171, j3=45.616, j4=-4.001, j5=80.973, j6=-5.833}
  [439] = {j1=-10.898, j2=64.699, j3=46.022, j4=-3.930, j5=80.631, j6=-6.270}
  [440] = {j1=-10.900, j2=64.614, j3=46.097, j4=-3.922, j5=80.567, j6=-6.345}
  [441] = {j1=-10.916, j2=64.135, j3=46.513, j4=-3.879, j5=80.217, j6=-6.772}
  [442] = {j1=-10.935, j2=63.657, j3=46.926, j4=-3.829, j5=79.877, j6=-7.196}
  [443] = {j1=-10.954, j2=63.181, j3=47.335, j4=-3.776, j5=79.548, j6=-7.614}
  [444] = {j1=-10.975, j2=62.707, j3=47.740, j4=-3.721, j5=79.232, j6=-8.025}
  [445] = {j1=-10.997, j2=62.235, j3=48.140, j4=-3.665, j5=78.928, j6=-8.427}
  [446] = {j1=-11.019, j2=61.766, j3=48.535, j4=-3.611, j5=78.640, j6=-8.816}
  [447] = {j1=-11.041, j2=61.300, j3=48.925, j4=-3.559, j5=78.367, j6=-9.193}
  [448] = {j1=-11.058, j2=60.896, j3=49.261, j4=-3.525, j5=78.141, j6=-9.504}
  [449] = {j1=-11.070, j2=60.497, j3=49.587, j4=-3.509, j5=77.933, j6=-9.791}
  [450] = {j1=-11.077, j2=60.106, j3=49.900, j4=-3.508, j5=77.747, j6=-10.054}
  [451] = {j1=-11.079, j2=59.727, j3=50.191, j4=-3.522, j5=77.587, j6=-10.290}
  [452] = {j1=-11.080, j2=59.712, j3=50.203, j4=-3.522, j5=77.580, j6=-10.298}
  [453] = {j1=-11.081, j2=59.765, j3=50.110, j4=-3.514, j5=77.713, j6=-10.215}
  [454] = {j1=-11.081, j2=59.777, j3=50.102, j4=-3.513, j5=77.716, j6=-10.207}
  [455] = {j1=-11.079, j2=60.156, j3=49.811, j4=-3.498, j5=77.876, j6=-9.968}
  [456] = {j1=-11.072, j2=60.546, j3=49.500, j4=-3.498, j5=78.062, j6=-9.703}
  [457] = {j1=-11.060, j2=60.944, j3=49.175, j4=-3.514, j5=78.268, j6=-9.414}
  [458] = {j1=-11.044, j2=61.347, j3=48.843, j4=-3.548, j5=78.489, j6=-9.102}
  [459] = {j1=-11.022, j2=61.809, j3=48.460, j4=-3.600, j5=78.755, j6=-8.727}
  [460] = {j1=-11.000, j2=62.273, j3=48.074, j4=-3.653, j5=79.034, j6=-8.341}
  [461] = {j1=-10.978, j2=62.738, j3=47.684, j4=-3.708, j5=79.325, j6=-7.944}
  [462] = {j1=-10.958, j2=63.207, j3=47.290, j4=-3.763, j5=79.630, j6=-7.537}
  [463] = {j1=-10.938, j2=63.677, j3=46.891, j4=-3.815, j5=79.948, j6=-7.122}
  [464] = {j1=-10.920, j2=64.151, j3=46.485, j4=-3.864, j5=80.280, j6=-6.701}
  [465] = {j1=-10.905, j2=64.629, j3=46.072, j4=-3.907, j5=80.626, j6=-6.274}
  [466] = {j1=-10.902, j2=64.711, j3=46.001, j4=-3.914, j5=80.685, j6=-6.199}
  [467] = {j1=-10.879, j2=65.183, j3=45.595, j4=-3.985, j5=81.028, j6=-5.758}
  [468] = {j1=-10.839, j2=65.707, j3=45.175, j4=-4.128, j5=81.362, j6=-5.248}
  [469] = {j1=-10.787, j2=66.161, j3=44.884, j4=-4.332, j5=81.540, j6=-4.795}
  [470] = {j1=-10.741, j2=66.463, j3=44.774, j4=-4.520, j5=81.526, j6=-4.509}
  [471] = {j1=-10.698, j2=66.705, j3=44.772, j4=-4.707, j5=81.378, j6=-4.305}
  [472] = {j1=-10.657, j2=66.897, j3=44.856, j4=-4.897, j5=81.118, j6=-4.169}
  [473] = {j1=-10.616, j2=67.050, j3=45.008, j4=-5.093, j5=80.768, j6=-4.087}
  [474] = {j1=-10.575, j2=67.172, j3=45.210, j4=-5.300, j5=80.348, j6=-4.044}
  [475] = {j1=-10.531, j2=67.271, j3=45.445, j4=-5.521, j5=79.880, j6=-4.027}
  [476] = {j1=-10.531, j2=67.286, j3=45.420, j4=-5.524, j5=79.927, j6=-3.991}
  [477] = {j1=-10.574, j2=67.185, j3=45.186, j4=-5.302, j5=80.391, j6=-4.009}
  [478] = {j1=-10.616, j2=67.062, j3=44.987, j4=-5.094, j5=80.807, j6=-4.052}
  [479] = {j1=-10.657, j2=66.908, j3=44.838, j4=-4.897, j5=81.153, j6=-4.134}
  [480] = {j1=-10.699, j2=66.713, j3=44.757, j4=-4.706, j5=81.408, j6=-4.271}
  [481] = {j1=-10.742, j2=66.469, j3=44.763, j4=-4.517, j5=81.551, j6=-4.476}
  [482] = {j1=-10.788, j2=66.165, j3=44.877, j4=-4.327, j5=81.560, j6=-4.764}
  [483] = {j1=-10.841, j2=65.708, j3=45.174, j4=-4.122, j5=81.374, j6=-5.218}
  [484] = {j1=-10.881, j2=65.181, j3=45.599, j4=-3.978, j5=81.033, j6=-5.731}
  [485] = {j1=-10.904, j2=64.706, j3=46.010, j4=-3.906, j5=80.684, j6=-6.173}
  [486] = {j1=-10.907, j2=64.621, j3=46.085, j4=-3.898, j5=80.620, j6=-6.249}
  [487] = {j1=-10.923, j2=64.142, j3=46.501, j4=-3.855, j5=80.271, j6=-6.675}
  [488] = {j1=-10.941, j2=63.667, j3=46.909, j4=-3.806, j5=79.936, j6=-7.096}
  [489] = {j1=-10.960, j2=63.195, j3=47.311, j4=-3.754, j5=79.615, j6=-7.509}
  [490] = {j1=-10.981, j2=62.726, j3=47.706, j4=-3.699, j5=79.309, j6=-7.914}
  [491] = {j1=-11.003, j2=62.260, j3=48.097, j4=-3.643, j5=79.015, j6=-8.310}
  [492] = {j1=-11.025, j2=61.795, j3=48.485, j4=-3.589, j5=78.734, j6=-8.696}
  [493] = {j1=-11.047, j2=61.331, j3=48.871, j4=-3.537, j5=78.465, j6=-9.070}
  [494] = {j1=-11.064, j2=60.926, j3=49.208, j4=-3.502, j5=78.239, j6=-9.382}
  [495] = {j1=-11.076, j2=60.525, j3=49.537, j4=-3.486, j5=78.027, j6=-9.673}
  [496] = {j1=-11.083, j2=60.132, j3=49.854, j4=-3.486, j5=77.835, j6=-9.938}
  [497] = {j1=-11.085, j2=59.750, j3=50.150, j4=-3.500, j5=77.669, j6=-10.177}
  [498] = {j1=-11.085, j2=59.736, j3=50.162, j4=-3.501, j5=77.662, j6=-10.186}
  [499] = {j1=-11.086, j2=59.754, j3=50.129, j4=-3.498, j5=77.709, j6=-10.155}
  [500] = {j1=-11.086, j2=59.767, j3=50.121, j4=-3.497, j5=77.712, j6=-10.147}
  [501] = {j1=-11.084, j2=60.147, j3=49.828, j4=-3.481, j5=77.874, j6=-9.907}
  [502] = {j1=-11.077, j2=60.538, j3=49.514, j4=-3.481, j5=78.063, j6=-9.640}
  [503] = {j1=-11.065, j2=60.937, j3=49.188, j4=-3.497, j5=78.272, j6=-9.350}
  [504] = {j1=-11.049, j2=61.340, j3=48.856, j4=-3.531, j5=78.493, j6=-9.037}
  [505] = {j1=-11.026, j2=61.801, j3=48.474, j4=-3.583, j5=78.757, j6=-8.663}
  [506] = {j1=-11.005, j2=62.263, j3=48.092, j4=-3.637, j5=79.031, j6=-8.279}
  [507] = {j1=-10.983, j2=62.726, j3=47.707, j4=-3.692, j5=79.317, j6=-7.885}
  [508] = {j1=-10.963, j2=63.191, j3=47.318, j4=-3.746, j5=79.617, j6=-7.481}
  [509] = {j1=-10.943, j2=63.660, j3=46.922, j4=-3.798, j5=79.930, j6=-7.069}
  [510] = {j1=-10.925, j2=64.132, j3=46.519, j4=-3.846, j5=80.259, j6=-6.650}
  [511] = {j1=-10.910, j2=64.609, j3=46.107, j4=-3.889, j5=80.604, j6=-6.223}
  [512] = {j1=-10.907, j2=64.692, j3=46.035, j4=-3.896, j5=80.664, j6=-6.148}
  [513] = {j1=-10.884, j2=65.166, j3=45.626, j4=-3.967, j5=81.010, j6=-5.705}
  [514] = {j1=-10.844, j2=65.692, j3=45.203, j4=-4.111, j5=81.349, j6=-5.189}
  [515] = {j1=-10.790, j2=66.149, j3=44.906, j4=-4.318, j5=81.534, j6=-4.732}
  [516] = {j1=-10.744, j2=66.451, j3=44.795, j4=-4.508, j5=81.522, j6=-4.443}
  [517] = {j1=-10.701, j2=66.694, j3=44.791, j4=-4.698, j5=81.376, j6=-4.236}
  [518] = {j1=-10.659, j2=66.887, j3=44.874, j4=-4.889, j5=81.117, j6=-4.099}
  [519] = {j1=-10.618, j2=67.040, j3=45.026, j4=-5.087, j5=80.766, j6=-4.015}
  [520] = {j1=-10.576, j2=67.162, j3=45.229, j4=-5.294, j5=80.347, j6=-3.972}
  [521] = {j1=-10.533, j2=67.261, j3=45.464, j4=-5.517, j5=79.878, j6=-3.954}
  [522] = {j1=-10.532, j2=67.286, j3=45.422, j4=-5.521, j5=79.955, j6=-3.896}
  [523] = {j1=-10.576, j2=67.185, j3=45.188, j4=-5.297, j5=80.419, j6=-3.915}
  [524] = {j1=-10.618, j2=67.062, j3=44.989, j4=-5.088, j5=80.835, j6=-3.959}
  [525] = {j1=-10.659, j2=66.907, j3=44.840, j4=-4.889, j5=81.180, j6=-4.043}
  [526] = {j1=-10.701, j2=66.712, j3=44.759, j4=-4.696, j5=81.435, j6=-4.182}
  [527] = {j1=-10.745, j2=66.467, j3=44.767, j4=-4.505, j5=81.575, j6=-4.389}
  [528] = {j1=-10.792, j2=66.162, j3=44.884, j4=-4.312, j5=81.580, j6=-4.681}
  [529] = {j1=-10.846, j2=65.701, j3=45.187, j4=-4.103, j5=81.387, j6=-5.142}
  [530] = {j1=-10.887, j2=65.171, j3=45.617, j4=-3.957, j5=81.038, j6=-5.661}
  [531] = {j1=-10.910, j2=64.694, j3=46.032, j4=-3.885, j5=80.685, j6=-6.106}
  [532] = {j1=-10.913, j2=64.609, j3=46.107, j4=-3.878, j5=80.621, j6=-6.181}
  [533] = {j1=-10.928, j2=64.131, j3=46.523, j4=-3.835, j5=80.271, j6=-6.608}
  [534] = {j1=-10.946, j2=63.657, j3=46.927, j4=-3.787, j5=79.940, j6=-7.026}
  [535] = {j1=-10.966, j2=63.188, j3=47.324, j4=-3.734, j5=79.625, j6=-7.436}
  [536] = {j1=-10.986, j2=62.723, j3=47.713, j4=-3.680, j5=79.326, j6=-7.837}
  [537] = {j1=-11.008, j2=62.259, j3=48.098, j4=-3.624, j5=79.039, j6=-8.229}
  [538] = {j1=-11.030, j2=61.797, j3=48.482, j4=-3.570, j5=78.763, j6=-8.611}
  [539] = {j1=-11.052, j2=61.334, j3=48.865, j4=-3.517, j5=78.497, j6=-8.984}
  [540] = {j1=-11.069, j2=60.930, j3=49.202, j4=-3.482, j5=78.270, j6=-9.297}
  [541] = {j1=-11.081, j2=60.528, j3=49.534, j4=-3.466, j5=78.055, j6=-9.589}
  [542] = {j1=-11.088, j2=60.133, j3=49.853, j4=-3.466, j5=77.859, j6=-9.857}
  [543] = {j1=-11.090, j2=59.749, j3=50.152, j4=-3.481, j5=77.690, j6=-10.099}
  [544] = {j1=-11.090, j2=59.734, j3=50.165, j4=-3.481, j5=77.682, j6=-10.107}
  [545] = {j1=-11.091, j2=59.765, j3=50.110, j4=-3.477, j5=77.761, j6=-10.057}
  [546] = {j1=-11.091, j2=59.778, j3=50.102, j4=-3.475, j5=77.764, j6=-10.049}
  [547] = {j1=-11.089, j2=60.160, j3=49.805, j4=-3.459, j5=77.930, j6=-9.806}
  [548] = {j1=-11.083, j2=60.553, j3=49.489, j4=-3.459, j5=78.123, j6=-9.537}
  [549] = {j1=-11.071, j2=60.953, j3=49.160, j4=-3.475, j5=78.335, j6=-9.244}
  [550] = {j1=-11.054, j2=61.356, j3=48.828, j4=-3.509, j5=78.556, j6=-8.931}
  [551] = {j1=-11.032, j2=61.815, j3=48.450, j4=-3.561, j5=78.816, j6=-8.559}
  [552] = {j1=-11.010, j2=62.273, j3=48.074, j4=-3.616, j5=79.083, j6=-8.178}
  [553] = {j1=-10.989, j2=62.732, j3=47.697, j4=-3.671, j5=79.361, j6=-7.788}
  [554] = {j1=-10.968, j2=63.193, j3=47.315, j4=-3.725, j5=79.652, j6=-7.390}
  [555] = {j1=-10.949, j2=63.658, j3=46.926, j4=-3.776, j5=79.958, j6=-6.983}
  [556] = {j1=-10.932, j2=64.128, j3=46.528, j4=-3.824, j5=80.282, j6=-6.566}
  [557] = {j1=-10.916, j2=64.604, j3=46.116, j4=-3.865, j5=80.626, j6=-6.140}
  [558] = {j1=-10.913, j2=64.687, j3=46.045, j4=-3.873, j5=80.686, j6=-6.064}
  [559] = {j1=-10.891, j2=65.162, j3=45.633, j4=-3.944, j5=81.036, j6=-5.617}
  [560] = {j1=-10.849, j2=65.692, j3=45.203, j4=-4.090, j5=81.384, j6=-5.095}
  [561] = {j1=-10.795, j2=66.153, j3=44.900, j4=-4.301, j5=81.577, j6=-4.630}
  [562] = {j1=-10.748, j2=66.457, j3=44.786, j4=-4.495, j5=81.570, j6=-4.336}
  [563] = {j1=-10.703, j2=66.701, j3=44.780, j4=-4.687, j5=81.426, j6=-4.126}
  [564] = {j1=-10.661, j2=66.894, j3=44.863, j4=-4.882, j5=81.168, j6=-3.986}
  [565] = {j1=-10.620, j2=67.047, j3=45.016, j4=-5.081, j5=80.818, j6=-3.901}
  [566] = {j1=-10.577, j2=67.168, j3=45.218, j4=-5.291, j5=80.398, j6=-3.856}
  [567] = {j1=-10.533, j2=67.268, j3=45.454, j4=-5.515, j5=79.930, j6=-3.837}
  [568] = {j1=-10.532, j2=67.292, j3=45.412, j4=-5.519, j5=80.007, j6=-3.780}
  [569] = {j1=-10.577, j2=67.191, j3=45.179, j4=-5.294, j5=80.470, j6=-3.799}
  [570] = {j1=-10.619, j2=67.068, j3=44.979, j4=-5.083, j5=80.885, j6=-3.845}
  [571] = {j1=-10.661, j2=66.913, j3=44.830, j4=-4.882, j5=81.230, j6=-3.931}
  [572] = {j1=-10.704, j2=66.718, j3=44.751, j4=-4.686, j5=81.482, j6=-4.072}
  [573] = {j1=-10.748, j2=66.472, j3=44.760, j4=-4.491, j5=81.620, j6=-4.283}
  [574] = {j1=-10.796, j2=66.165, j3=44.880, j4=-4.294, j5=81.620, j6=-4.580}
  [575] = {j1=-10.852, j2=65.700, j3=45.189, j4=-4.082, j5=81.418, j6=-5.049}
  [576] = {j1=-10.893, j2=65.166, j3=45.626, j4=-3.934, j5=81.062, j6=-5.574}
  [577] = {j1=-10.916, j2=64.688, j3=46.044, j4=-3.862, j5=80.704, j6=-6.022}
  [578] = {j1=-10.919, j2=64.603, j3=46.119, j4=-3.854, j5=80.639, j6=-6.098}
  [579] = {j1=-10.935, j2=64.125, j3=46.534, j4=-3.812, j5=80.290, j6=-6.524}
  [580] = {j1=-10.952, j2=63.653, j3=46.935, j4=-3.764, j5=79.963, j6=-6.939}
  [581] = {j1=-10.972, j2=63.188, j3=47.325, j4=-3.713, j5=79.656, j6=-7.344}
  [582] = {j1=-10.992, j2=62.726, j3=47.707, j4=-3.658, j5=79.364, j6=-7.740}
  [583] = {j1=-11.014, j2=62.267, j3=48.086, j4=-3.603, j5=79.086, j6=-8.128}
  [584] = {j1=-11.036, j2=61.808, j3=48.463, j4=-3.548, j5=78.817, j6=-8.507}
  [585] = {j1=-11.058, j2=61.347, j3=48.843, j4=-3.495, j5=78.553, j6=-8.879}
  [586] = {j1=-11.075, j2=60.942, j3=49.180, j4=-3.459, j5=78.326, j6=-9.192}
  [587] = {j1=-11.087, j2=60.539, j3=49.514, j4=-3.443, j5=78.109, j6=-9.486}
  [588] = {j1=-11.094, j2=60.143, j3=49.836, j4=-3.443, j5=77.908, j6=-9.757}
  [589] = {j1=-11.096, j2=59.757, j3=50.139, j4=-3.459, j5=77.734, j6=-10.000}
  [590] = {j1=-11.096, j2=59.742, j3=50.152, j4=-3.460, j5=77.726, j6=-10.009}
  [591] = {j1=-11.097, j2=59.773, j3=50.097, j4=-3.455, j5=77.805, j6=-9.958}
  [592] = {j1=-11.097, j2=59.786, j3=50.088, j4=-3.453, j5=77.808, j6=-9.950}
  [593] = {j1=-11.095, j2=60.170, j3=49.789, j4=-3.437, j5=77.979, j6=-9.705}
  [594] = {j1=-11.089, j2=60.564, j3=49.470, j4=-3.436, j5=78.175, j6=-9.434}
  [595] = {j1=-11.077, j2=60.965, j3=49.140, j4=-3.452, j5=78.389, j6=-9.139}
  [596] = {j1=-11.060, j2=61.367, j3=48.808, j4=-3.487, j5=78.610, j6=-8.826}
  [597] = {j1=-11.038, j2=61.824, j3=48.434, j4=-3.540, j5=78.866, j6=-8.454}
  [598] = {j1=-11.016, j2=62.279, j3=48.064, j4=-3.594, j5=79.127, j6=-8.077}
  [599] = {j1=-10.995, j2=62.734, j3=47.694, j4=-3.649, j5=79.396, j6=-7.692}
  [600] = {j1=-10.974, j2=63.191, j3=47.319, j4=-3.702, j5=79.679, j6=-7.299}
  [601] = {j1=-10.955, j2=63.653, j3=46.937, j4=-3.754, j5=79.977, j6=-6.895}
  [602] = {j1=-10.938, j2=64.120, j3=46.542, j4=-3.800, j5=80.297, j6=-6.481}
  [603] = {j1=-10.923, j2=64.596, j3=46.132, j4=-3.841, j5=80.640, j6=-6.056}
  [604] = {j1=-10.920, j2=64.679, j3=46.061, j4=-3.848, j5=80.700, j6=-5.980}
  [605] = {j1=-10.897, j2=65.155, j3=45.646, j4=-3.920, j5=81.054, j6=-5.531}
  [606] = {j1=-10.855, j2=65.688, j3=45.210, j4=-4.068, j5=81.410, j6=-5.002}
  [607] = {j1=-10.799, j2=66.152, j3=44.902, j4=-4.282, j5=81.610, j6=-4.530}
  [608] = {j1=-10.751, j2=66.459, j3=44.785, j4=-4.481, j5=81.607, j6=-4.230}
  [609] = {j1=-10.706, j2=66.703, j3=44.778, j4=-4.676, j5=81.466, j6=-4.017}
  [610] = {j1=-10.663, j2=66.897, j3=44.860, j4=-4.873, j5=81.209, j6=-3.874}
  [611] = {j1=-10.621, j2=67.050, j3=45.012, j4=-5.075, j5=80.860, j6=-3.787}
  [612] = {j1=-10.579, j2=67.171, j3=45.215, j4=-5.286, j5=80.442, j6=-3.741}
  [613] = {j1=-10.534, j2=67.271, j3=45.451, j4=-5.512, j5=79.974, j6=-3.720}
  [614] = {j1=-10.533, j2=67.297, j3=45.406, j4=-5.516, j5=80.056, j6=-3.659}
  [615] = {j1=-10.578, j2=67.196, j3=45.173, j4=-5.290, j5=80.518, j6=-3.680}
  [616] = {j1=-10.621, j2=67.072, j3=44.974, j4=-5.077, j5=80.931, j6=-3.727}
  [617] = {j1=-10.663, j2=66.917, j3=44.825, j4=-4.873, j5=81.274, j6=-3.816}
  [618] = {j1=-10.707, j2=66.721, j3=44.747, j4=-4.674, j5=81.525, j6=-3.960}
  [619] = {j1=-10.752, j2=66.474, j3=44.759, j4=-4.477, j5=81.660, j6=-4.175}
  [620] = {j1=-10.801, j2=66.164, j3=44.882, j4=-4.276, j5=81.654, j6=-4.477}
  [621] = {j1=-10.858, j2=65.696, j3=45.197, j4=-4.059, j5=81.446, j6=-4.953}
  [622] = {j1=-10.900, j2=65.160, j3=45.639, j4=-3.909, j5=81.081, j6=-5.484}
  [623] = {j1=-10.923, j2=64.680, j3=46.060, j4=-3.836, j5=80.720, j6=-5.935}
  [624] = {j1=-10.926, j2=64.594, j3=46.135, j4=-3.829, j5=80.654, j6=-6.011}
  [625] = {j1=-10.942, j2=64.117, j3=46.549, j4=-3.788, j5=80.306, j6=-6.436}
  [626] = {j1=-10.959, j2=63.648, j3=46.946, j4=-3.741, j5=79.984, j6=-6.848}
  [627] = {j1=-10.978, j2=63.186, j3=47.330, j4=-3.690, j5=79.683, j6=-7.250}
  [628] = {j1=-10.998, j2=62.728, j3=47.705, j4=-3.636, j5=79.400, j6=-7.641}
  [629] = {j1=-11.020, j2=62.273, j3=48.077, j4=-3.580, j5=79.129, j6=-8.024}
  [630] = {j1=-11.042, j2=61.817, j3=48.448, j4=-3.525, j5=78.866, j6=-8.399}
  [631] = {j1=-11.064, j2=61.358, j3=48.825, j4=-3.471, j5=78.606, j6=-8.770}
  [632] = {j1=-11.082, j2=60.953, j3=49.162, j4=-3.435, j5=78.379, j6=-9.084}
  [633] = {j1=-11.094, j2=60.549, j3=49.497, j4=-3.419, j5=78.159, j6=-9.379}
  [634] = {j1=-11.101, j2=60.151, j3=49.822, j4=-3.419, j5=77.956, j6=-9.652}
  [635] = {j1=-11.103, j2=59.764, j3=50.128, j4=-3.436, j5=77.777, j6=-9.898}
  [636] = {j1=-11.103, j2=59.748, j3=50.141, j4=-3.436, j5=77.769, j6=-9.906}
  [637] = {j1=-11.104, j2=59.782, j3=50.082, j4=-3.431, j5=77.854, j6=-9.852}
  [638] = {j1=-11.104, j2=59.795, j3=50.073, j4=-3.430, j5=77.857, j6=-9.843}
  [639] = {j1=-11.102, j2=60.180, j3=49.771, j4=-3.412, j5=78.032, j6=-9.597}
  [640] = {j1=-11.095, j2=60.576, j3=49.450, j4=-3.411, j5=78.231, j6=-9.323}
  [641] = {j1=-11.083, j2=60.977, j3=49.119, j4=-3.427, j5=78.446, j6=-9.027}
  [642] = {j1=-11.066, j2=61.379, j3=48.788, j4=-3.463, j5=78.667, j6=-8.713}
  [643] = {j1=-11.044, j2=61.834, j3=48.418, j4=-3.516, j5=78.919, j6=-8.344}
  [644] = {j1=-11.022, j2=62.285, j3=48.054, j4=-3.571, j5=79.173, j6=-7.970}
  [645] = {j1=-11.001, j2=62.736, j3=47.691, j4=-3.626, j5=79.434, j6=-7.589}
  [646] = {j1=-10.981, j2=63.189, j3=47.324, j4=-3.679, j5=79.708, j6=-7.200}
  [647] = {j1=-10.962, j2=63.647, j3=46.947, j4=-3.729, j5=80.000, j6=-6.801}
  [648] = {j1=-10.945, j2=64.112, j3=46.557, j4=-3.775, j5=80.314, j6=-6.390}
  [649] = {j1=-10.930, j2=64.587, j3=46.149, j4=-3.815, j5=80.656, j6=-5.966}
  [650] = {j1=-10.927, j2=64.670, j3=46.078, j4=-3.822, j5=80.716, j6=-5.890}
  [651] = {j1=-10.904, j2=65.148, j3=45.660, j4=-3.894, j5=81.073, j6=-5.438}
  [652] = {j1=-10.862, j2=65.683, j3=45.220, j4=-4.044, j5=81.435, j6=-4.903}
  [653] = {j1=-10.805, j2=66.150, j3=44.907, j4=-4.263, j5=81.642, j6=-4.424}
  [654] = {j1=-10.755, j2=66.458, j3=44.786, j4=-4.465, j5=81.644, j6=-4.119}
  [655] = {j1=-10.709, j2=66.704, j3=44.777, j4=-4.664, j5=81.506, j6=-3.902}
  [656] = {j1=-10.666, j2=66.899, j3=44.858, j4=-4.864, j5=81.252, j6=-3.756}
  [657] = {j1=-10.623, j2=67.052, j3=45.010, j4=-5.068, j5=80.904, j6=-3.666}
  [658] = {j1=-10.580, j2=67.174, j3=45.212, j4=-5.282, j5=80.487, j6=-3.618}
  [659] = {j1=-10.535, j2=67.274, j3=45.447, j4=-5.509, j5=80.021, j6=-3.595}
  [660] = {j1=-10.534, j2=67.299, j3=45.403, j4=-5.513, j5=80.102, j6=-3.534}
  [661] = {j1=-10.579, j2=67.198, j3=45.171, j4=-5.285, j5=80.562, j6=-3.557}
  [662] = {j1=-10.623, j2=67.074, j3=44.972, j4=-5.070, j5=80.973, j6=-3.607}
  [663] = {j1=-10.666, j2=66.918, j3=44.825, j4=-4.864, j5=81.314, j6=-3.698}
  [664] = {j1=-10.710, j2=66.721, j3=44.748, j4=-4.662, j5=81.562, j6=-3.845}
  [665] = {j1=-10.756, j2=66.472, j3=44.763, j4=-4.461, j5=81.693, j6=-4.064}
  [666] = {j1=-10.806, j2=66.161, j3=44.889, j4=-4.256, j5=81.683, j6=-4.372}
  [667] = {j1=-10.864, j2=65.690, j3=45.209, j4=-4.034, j5=81.467, j6=-4.854}
  [668] = {j1=-10.907, j2=65.150, j3=45.656, j4=-3.882, j5=81.097, j6=-5.391}
  [669] = {j1=-10.931, j2=64.669, j3=46.079, j4=-3.810, j5=80.732, j6=-5.844}
  [670] = {j1=-10.933, j2=64.584, j3=46.155, j4=-3.802, j5=80.666, j6=-5.920}
  [671] = {j1=-10.949, j2=64.107, j3=46.567, j4=-3.763, j5=80.319, j6=-6.344}
  [672] = {j1=-10.966, j2=63.640, j3=46.960, j4=-3.716, j5=80.001, j6=-6.754}
  [673] = {j1=-10.985, j2=63.181, j3=47.338, j4=-3.666, j5=79.707, j6=-7.151}
  [674] = {j1=-11.005, j2=62.727, j3=47.707, j4=-3.612, j5=79.431, j6=-7.538}
  [675] = {j1=-11.026, j2=62.276, j3=48.072, j4=-3.556, j5=79.168, j6=-7.916}
  [676] = {j1=-11.048, j2=61.823, j3=48.438, j4=-3.501, j5=78.911, j6=-8.289}
  [677] = {j1=-11.071, j2=61.366, j3=48.812, j4=-3.446, j5=78.655, j6=-8.658}
  [678] = {j1=-11.088, j2=60.962, j3=49.147, j4=-3.410, j5=78.429, j6=-8.972}
  [679] = {j1=-11.100, j2=60.557, j3=49.484, j4=-3.393, j5=78.207, j6=-9.269}
  [680] = {j1=-11.107, j2=60.157, j3=49.811, j4=-3.394, j5=78.000, j6=-9.543}
  [681] = {j1=-11.109, j2=59.769, j3=50.120, j4=-3.411, j5=77.818, j6=-9.791}
  [682] = {j1=-11.109, j2=59.753, j3=50.134, j4=-3.412, j5=77.809, j6=-9.800}
  [683] = {j1=-11.110, j2=59.787, j3=50.074, j4=-3.406, j5=77.895, j6=-9.745}
  [684] = {j1=-11.110, j2=59.800, j3=50.066, j4=-3.405, j5=77.898, j6=-9.736}
  [685] = {j1=-11.109, j2=60.186, j3=49.761, j4=-3.387, j5=78.075, j6=-9.488}
  [686] = {j1=-11.102, j2=60.583, j3=49.438, j4=-3.385, j5=78.277, j6=-9.213}
  [687] = {j1=-11.090, j2=60.985, j3=49.107, j4=-3.401, j5=78.493, j6=-8.916}
  [688] = {j1=-11.073, j2=61.386, j3=48.777, j4=-3.437, j5=78.713, j6=-8.601}
  [689] = {j1=-11.050, j2=61.838, j3=48.411, j4=-3.492, j5=78.960, j6=-8.233}
  [690] = {j1=-11.028, j2=62.287, j3=48.053, j4=-3.547, j5=79.208, j6=-7.862}
  [691] = {j1=-11.007, j2=62.734, j3=47.696, j4=-3.602, j5=79.462, j6=-7.486}
  [692] = {j1=-10.987, j2=63.183, j3=47.336, j4=-3.655, j5=79.728, j6=-7.102}
  [693] = {j1=-10.969, j2=63.638, j3=46.965, j4=-3.704, j5=80.013, j6=-6.706}
  [694] = {j1=-10.952, j2=64.100, j3=46.579, j4=-3.749, j5=80.323, j6=-6.298}
  [695] = {j1=-10.937, j2=64.574, j3=46.173, j4=-3.788, j5=80.663, j6=-5.875}
  [696] = {j1=-10.935, j2=64.657, j3=46.102, j4=-3.795, j5=80.723, j6=-5.799}
  [697] = {j1=-10.912, j2=65.136, j3=45.683, j4=-3.867, j5=81.082, j6=-5.345}
  [698] = {j1=-10.868, j2=65.674, j3=45.238, j4=-4.019, j5=81.450, j6=-4.806}
  [699] = {j1=-10.810, j2=66.143, j3=44.921, j4=-4.242, j5=81.663, j6=-4.319}
  [700] = {j1=-10.760, j2=66.453, j3=44.797, j4=-4.449, j5=81.669, j6=-4.010}
  [701] = {j1=-10.713, j2=66.700, j3=44.786, j4=-4.651, j5=81.534, j6=-3.788}
  [702] = {j1=-10.669, j2=66.895, j3=44.865, j4=-4.854, j5=81.282, j6=-3.639}
  [703] = {j1=-10.625, j2=67.050, j3=45.015, j4=-5.061, j5=80.937, j6=-3.546}
  [704] = {j1=-10.582, j2=67.172, j3=45.217, j4=-5.276, j5=80.521, j6=-3.495}
  [705] = {j1=-10.537, j2=67.273, j3=45.451, j4=-5.505, j5=80.058, j6=-3.470}
  [706] = {j1=-10.536, j2=67.298, j3=45.407, j4=-5.509, j5=80.139, j6=-3.409}
  [707] = {j1=-10.581, j2=67.195, j3=45.177, j4=-5.279, j5=80.596, j6=-3.435}
  [708] = {j1=-10.625, j2=67.070, j3=44.980, j4=-5.062, j5=81.004, j6=-3.487}
  [709] = {j1=-10.669, j2=66.913, j3=44.835, j4=-4.853, j5=81.342, j6=-3.581}
  [710] = {j1=-10.714, j2=66.715, j3=44.760, j4=-4.649, j5=81.586, j6=-3.732}
  [711] = {j1=-10.761, j2=66.465, j3=44.777, j4=-4.444, j5=81.714, j6=-3.956}
  [712] = {j1=-10.812, j2=66.151, j3=44.907, j4=-4.235, j5=81.700, j6=-4.268}
  [713] = {j1=-10.871, j2=65.678, j3=45.231, j4=-4.009, j5=81.478, j6=-4.757}
  [714] = {j1=-10.915, j2=65.136, j3=45.682, j4=-3.855, j5=81.102, j6=-5.299}
  [715] = {j1=-10.938, j2=64.654, j3=46.106, j4=-3.782, j5=80.735, j6=-5.753}
  [716] = {j1=-10.941, j2=64.569, j3=46.182, j4=-3.775, j5=80.669, j6=-5.829}
  [717] = {j1=-10.956, j2=64.093, j3=46.593, j4=-3.736, j5=80.324, j6=-6.252}
  [718] = {j1=-10.973, j2=63.628, j3=46.982, j4=-3.691, j5=80.010, j6=-6.659}
  [719] = {j1=-10.991, j2=63.173, j3=47.355, j4=-3.641, j5=79.722, j6=-7.052}
  [720] = {j1=-11.011, j2=62.722, j3=47.718, j4=-3.587, j5=79.452, j6=-7.435}
  [721] = {j1=-11.033, j2=62.273, j3=48.077, j4=-3.532, j5=79.195, j6=-7.809}
  [722] = {j1=-11.055, j2=61.823, j3=48.438, j4=-3.476, j5=78.944, j6=-8.179}
  [723] = {j1=-11.078, j2=61.368, j3=48.808, j4=-3.420, j5=78.692, j6=-8.547}
  [724] = {j1=-11.095, j2=60.965, j3=49.143, j4=-3.383, j5=78.466, j6=-8.861}
  [725] = {j1=-11.108, j2=60.560, j3=49.480, j4=-3.366, j5=78.244, j6=-9.159}
  [726] = {j1=-11.115, j2=60.159, j3=49.809, j4=-3.367, j5=78.034, j6=-9.435}
  [727] = {j1=-11.116, j2=59.769, j3=50.120, j4=-3.385, j5=77.849, j6=-9.684}
  [728] = {j1=-11.116, j2=59.753, j3=50.134, j4=-3.386, j5=77.840, j6=-9.692}
  [729] = {j1=-11.117, j2=59.788, j3=50.074, j4=-3.380, j5=77.926, j6=-9.637}
  [730] = {j1=-11.118, j2=59.800, j3=50.066, j4=-3.379, j5=77.929, j6=-9.629}
  [731] = {j1=-11.116, j2=60.187, j3=49.759, j4=-3.360, j5=78.108, j6=-9.379}
  [732] = {j1=-11.110, j2=60.585, j3=49.435, j4=-3.358, j5=78.312, j6=-9.103}
  [733] = {j1=-11.098, j2=60.986, j3=49.104, j4=-3.374, j5=78.528, j6=-8.805}
  [734] = {j1=-11.080, j2=61.387, j3=48.776, j4=-3.411, j5=78.746, j6=-8.491}
  [735] = {j1=-11.057, j2=61.837, j3=48.414, j4=-3.466, j5=78.990, j6=-8.124}
  [736] = {j1=-11.035, j2=62.283, j3=48.061, j4=-3.522, j5=79.232, j6=-7.756}
  [737] = {j1=-11.014, j2=62.727, j3=47.710, j4=-3.577, j5=79.479, j6=-7.383}
  [738] = {j1=-10.994, j2=63.172, j3=47.356, j4=-3.629, j5=79.738, j6=-7.002}
  [739] = {j1=-10.976, j2=63.624, j3=46.991, j4=-3.679, j5=80.017, j6=-6.611}
  [740] = {j1=-10.960, j2=64.084, j3=46.609, j4=-3.723, j5=80.322, j6=-6.206}
  [741] = {j1=-10.945, j2=64.557, j3=46.204, j4=-3.760, j5=80.660, j6=-5.784}
  [742] = {j1=-10.943, j2=64.639, j3=46.133, j4=-3.767, j5=80.720, j6=-5.708}
  [743] = {j1=-10.919, j2=65.119, j3=45.714, j4=-3.838, j5=81.081, j6=-5.253}
  [744] = {j1=-10.875, j2=65.658, j3=45.266, j4=-3.993, j5=81.452, j6=-4.709}
  [745] = {j1=-10.816, j2=66.130, j3=44.945, j4=-4.220, j5=81.670, j6=-4.217}
  [746] = {j1=-10.764, j2=66.441, j3=44.819, j4=-4.431, j5=81.680, j6=-3.902}
  [747] = {j1=-10.717, j2=66.690, j3=44.805, j4=-4.637, j5=81.548, j6=-3.676}
  [748] = {j1=-10.672, j2=66.887, j3=44.882, j4=-4.842, j5=81.300, j6=-3.523}
  [749] = {j1=-10.628, j2=67.042, j3=45.031, j4=-5.052, j5=80.958, j6=-3.427}
  [750] = {j1=-10.584, j2=67.166, j3=45.230, j4=-5.269, j5=80.545, j6=-3.373}
  [751] = {j1=-10.538, j2=67.267, j3=45.463, j4=-5.499, j5=80.084, j6=-3.345}
  [752] = {j1=-10.537, j2=67.292, j3=45.419, j4=-5.504, j5=80.164, j6=-3.284}
  [753] = {j1=-10.583, j2=67.188, j3=45.191, j4=-5.272, j5=80.618, j6=-3.313}
  [754] = {j1=-10.627, j2=67.062, j3=44.997, j4=-5.053, j5=81.023, j6=-3.368}
  [755] = {j1=-10.672, j2=66.903, j3=44.854, j4=-4.842, j5=81.357, j6=-3.466}
  [756] = {j1=-10.717, j2=66.703, j3=44.782, j4=-4.634, j5=81.597, j6=-3.621}
  [757] = {j1=-10.766, j2=66.451, j3=44.802, j4=-4.426, j5=81.721, j6=-3.849}
  [758] = {j1=-10.818, j2=66.136, j3=44.935, j4=-4.212, j5=81.703, j6=-4.166}
  [759] = {j1=-10.878, j2=65.661, j3=45.263, j4=-3.982, j5=81.476, j6=-4.661}
  [760] = {j1=-10.923, j2=65.118, j3=45.716, j4=-3.826, j5=81.097, j6=-5.206}
  [761] = {j1=-10.946, j2=64.635, j3=46.141, j4=-3.753, j5=80.728, j6=-5.662}
  [762] = {j1=-10.949, j2=64.550, j3=46.217, j4=-3.746, j5=80.662, j6=-5.738}
  [763] = {j1=-10.963, j2=64.075, j3=46.626, j4=-3.709, j5=80.318, j6=-6.159}
  [764] = {j1=-10.980, j2=63.612, j3=47.012, j4=-3.664, j5=80.008, j6=-6.563}
  [765] = {j1=-10.998, j2=63.159, j3=47.380, j4=-3.615, j5=79.725, j6=-6.953}
  [766] = {j1=-11.018, j2=62.711, j3=47.738, j4=-3.562, j5=79.462, j6=-7.332}
  [767] = {j1=-11.040, j2=62.265, j3=48.092, j4=-3.506, j5=79.211, j6=-7.703}
  [768] = {j1=-11.062, j2=61.818, j3=48.448, j4=-3.450, j5=78.965, j6=-8.070}
  [769] = {j1=-11.085, j2=61.365, j3=48.815, j4=-3.393, j5=78.716, j6=-8.436}
  [770] = {j1=-11.103, j2=60.962, j3=49.149, j4=-3.355, j5=78.492, j6=-8.751}
  [771] = {j1=-11.115, j2=60.557, j3=49.486, j4=-3.338, j5=78.269, j6=-9.049}
  [772] = {j1=-11.122, j2=60.156, j3=49.816, j4=-3.339, j5=78.058, j6=-9.326}
  [773] = {j1=-11.124, j2=59.764, j3=50.130, j4=-3.358, j5=77.870, j6=-9.576}
  [774] = {j1=-11.124, j2=59.748, j3=50.144, j4=-3.359, j5=77.860, j6=-9.585}
  [775] = {j1=-11.125, j2=59.783, j3=50.083, j4=-3.353, j5=77.946, j6=-9.529}
  [776] = {j1=-11.125, j2=59.795, j3=50.075, j4=-3.352, j5=77.949, j6=-9.521}
  [777] = {j1=-11.124, j2=60.183, j3=49.767, j4=-3.332, j5=78.131, j6=-9.270}
  [778] = {j1=-11.117, j2=60.581, j3=49.443, j4=-3.329, j5=78.335, j6=-8.993}
  [779] = {j1=-11.105, j2=60.982, j3=49.113, j4=-3.346, j5=78.550, j6=-8.695}
  [780] = {j1=-11.087, j2=61.381, j3=48.787, j4=-3.384, j5=78.767, j6=-8.381}
  [781] = {j1=-11.064, j2=61.830, j3=48.428, j4=-3.440, j5=79.006, j6=-8.015}
  [782] = {j1=-11.042, j2=62.273, j3=48.079, j4=-3.496, j5=79.243, j6=-7.650}
  [783] = {j1=-11.021, j2=62.714, j3=47.734, j4=-3.551, j5=79.484, j6=-7.280}
  [784] = {j1=-11.002, j2=63.157, j3=47.385, j4=-3.603, j5=79.737, j6=-6.903}
  [785] = {j1=-10.984, j2=63.605, j3=47.024, j4=-3.651, j5=80.011, j6=-6.514}
  [786] = {j1=-10.967, j2=64.064, j3=46.646, j4=-3.695, j5=80.312, j6=-6.112}
  [787] = {j1=-10.953, j2=64.535, j3=46.244, j4=-3.731, j5=80.647, j6=-5.692}
  [788] = {j1=-10.951, j2=64.617, j3=46.173, j4=-3.737, j5=80.707, j6=-5.616}
  [789] = {j1=-10.927, j2=65.096, j3=45.754, j4=-3.808, j5=81.068, j6=-5.160}
  [790] = {j1=-10.883, j2=65.637, j3=45.305, j4=-3.965, j5=81.442, j6=-4.613}
  [791] = {j1=-10.822, j2=66.110, j3=44.981, j4=-4.197, j5=81.663, j6=-4.116}
  [792] = {j1=-10.769, j2=66.423, j3=44.852, j4=-4.412, j5=81.676, j6=-3.796}
  [793] = {j1=-10.721, j2=66.673, j3=44.836, j4=-4.621, j5=81.548, j6=-3.566}
  [794] = {j1=-10.675, j2=66.872, j3=44.910, j4=-4.830, j5=81.303, j6=-3.408}
  [795] = {j1=-10.630, j2=67.029, j3=45.056, j4=-5.042, j5=80.965, j6=-3.309}
  [796] = {j1=-10.586, j2=67.154, j3=45.253, j4=-5.261, j5=80.556, j6=-3.251}
  [797] = {j1=-10.540, j2=67.256, j3=45.483, j4=-5.493, j5=80.098, j6=-3.220}
  [798] = {j1=-10.539, j2=67.281, j3=45.440, j4=-5.497, j5=80.178, j6=-3.159}
  [799] = {j1=-10.585, j2=67.176, j3=45.215, j4=-5.264, j5=80.627, j6=-3.191}
  [800] = {j1=-10.630, j2=67.047, j3=45.024, j4=-5.043, j5=81.028, j6=-3.251}
  [801] = {j1=-10.675, j2=66.887, j3=44.884, j4=-4.829, j5=81.357, j6=-3.352}
  [802] = {j1=-10.722, j2=66.685, j3=44.816, j4=-4.618, j5=81.593, j6=-3.512}
  [803] = {j1=-10.771, j2=66.431, j3=44.839, j4=-4.406, j5=81.713, j6=-3.744}
  [804] = {j1=-10.824, j2=66.114, j3=44.974, j4=-4.189, j5=81.691, j6=-4.066}
  [805] = {j1=-10.886, j2=65.637, j3=45.305, j4=-3.954, j5=81.461, j6=-4.565}
  [806] = {j1=-10.931, j2=65.093, j3=45.760, j4=-3.795, j5=81.079, j6=-5.114}
  [807] = {j1=-10.954, j2=64.611, j3=46.185, j4=-3.723, j5=80.711, j6=-5.570}
  [808] = {j1=-10.957, j2=64.525, j3=46.261, j4=-3.716, j5=80.644, j6=-5.645}
  [809] = {j1=-10.971, j2=64.051, j3=46.668, j4=-3.680, j5=80.302, j6=-6.065}
  [810] = {j1=-10.988, j2=63.591, j3=47.051, j4=-3.637, j5=79.996, j6=-6.466}
  [811] = {j1=-11.006, j2=63.140, j3=47.415, j4=-3.588, j5=79.717, j6=-6.853}
  [812] = {j1=-11.026, j2=62.694, j3=47.769, j4=-3.535, j5=79.459, j6=-7.229}
  [813] = {j1=-11.047, j2=62.251, j3=48.118, j4=-3.479, j5=79.213, j6=-7.597}
  [814] = {j1=-11.069, j2=61.806, j3=48.471, j4=-3.422, j5=78.972, j6=-7.962}
  [815] = {j1=-11.093, j2=61.354, j3=48.835, j4=-3.365, j5=78.726, j6=-8.327}
  [816] = {j1=-11.111, j2=60.952, j3=49.166, j4=-3.326, j5=78.503, j6=-8.641}
  [817] = {j1=-11.124, j2=60.548, j3=49.503, j4=-3.308, j5=78.280, j6=-8.940}
  [818] = {j1=-11.130, j2=60.146, j3=49.834, j4=-3.310, j5=78.068, j6=-9.217}
  [819] = {j1=-11.132, j2=59.754, j3=50.149, j4=-3.329, j5=77.878, j6=-9.468}
  [820] = {j1=-11.132, j2=59.738, j3=50.163, j4=-3.330, j5=77.868, j6=-9.477}
  [821] = {j1=-11.133, j2=59.772, j3=50.102, j4=-3.324, j5=77.955, j6=-9.421}
  [822] = {j1=-11.133, j2=59.784, j3=50.095, j4=-3.323, j5=77.957, j6=-9.412}
  [823] = {j1=-11.132, j2=60.173, j3=49.786, j4=-3.302, j5=78.140, j6=-9.161}
  [824] = {j1=-11.125, j2=60.571, j3=49.462, j4=-3.300, j5=78.344, j6=-8.884}
  [825] = {j1=-11.113, j2=60.971, j3=49.133, j4=-3.317, j5=78.559, j6=-8.586}
  [826] = {j1=-11.095, j2=61.369, j3=48.809, j4=-3.355, j5=78.773, j6=-8.272}
  [827] = {j1=-11.072, j2=61.816, j3=48.454, j4=-3.412, j5=79.009, j6=-7.908}
  [828] = {j1=-11.050, j2=62.256, j3=48.109, j4=-3.469, j5=79.240, j6=-7.544}
  [829] = {j1=-11.029, j2=62.695, j3=47.769, j4=-3.524, j5=79.476, j6=-7.177}
  [830] = {j1=-11.009, j2=63.135, j3=47.424, j4=-3.575, j5=79.724, j6=-6.803}
  [831] = {j1=-10.991, j2=63.581, j3=47.068, j4=-3.623, j5=79.993, j6=-6.417}
  [832] = {j1=-10.975, j2=64.038, j3=46.693, j4=-3.665, j5=80.290, j6=-6.017}
  [833] = {j1=-10.961, j2=64.507, j3=46.293, j4=-3.700, j5=80.623, j6=-5.599}
  [834] = {j1=-10.959, j2=64.589, j3=46.223, j4=-3.706, j5=80.682, j6=-5.523}
  [835] = {j1=-10.936, j2=65.068, j3=45.805, j4=-3.777, j5=81.042, j6=-5.068}
  [836] = {j1=-10.891, j2=65.609, j3=45.355, j4=-3.936, j5=81.417, j6=-4.518}
  [837] = {j1=-10.829, j2=66.083, j3=45.029, j4=-4.172, j5=81.641, j6=-4.016}
  [838] = {j1=-10.775, j2=66.398, j3=44.898, j4=-4.391, j5=81.657, j6=-3.692}
  [839] = {j1=-10.725, j2=66.650, j3=44.879, j4=-4.604, j5=81.533, j6=-3.457}
  [840] = {j1=-10.679, j2=66.850, j3=44.950, j4=-4.816, j5=81.292, j6=-3.295}
  [841] = {j1=-10.634, j2=67.009, j3=45.092, j4=-5.030, j5=80.957, j6=-3.191}
  [842] = {j1=-10.589, j2=67.136, j3=45.286, j4=-5.252, j5=80.552, j6=-3.130}
  [843] = {j1=-10.542, j2=67.240, j3=45.514, j4=-5.485, j5=80.099, j6=-3.095}
  [844] = {j1=-10.541, j2=67.265, j3=45.471, j4=-5.489, j5=80.178, j6=-3.035}
  [845] = {j1=-10.588, j2=67.157, j3=45.249, j4=-5.254, j5=80.622, j6=-3.070}
  [846] = {j1=-10.633, j2=67.027, j3=45.062, j4=-5.031, j5=81.018, j6=-3.134}
  [847] = {j1=-10.679, j2=66.864, j3=44.927, j4=-4.814, j5=81.342, j6=-3.240}
  [848] = {j1=-10.726, j2=66.660, j3=44.862, j4=-4.600, j5=81.574, j6=-3.404}
  [849] = {j1=-10.776, j2=66.404, j3=44.889, j4=-4.385, j5=81.688, j6=-3.641}
  [850] = {j1=-10.831, j2=66.085, j3=45.027, j4=-4.163, j5=81.663, j6=-3.967}
  [851] = {j1=-10.894, j2=65.607, j3=45.360, j4=-3.924, j5=81.430, j6=-4.471}
  [852] = {j1=-10.940, j2=65.063, j3=45.815, j4=-3.764, j5=81.048, j6=-5.021}
  [853] = {j1=-10.963, j2=64.581, j3=46.239, j4=-3.692, j5=80.680, j6=-5.477}
  [854] = {j1=-10.966, j2=64.495, j3=46.315, j4=-3.685, j5=80.614, j6=-5.552}
  [855] = {j1=-10.980, j2=64.022, j3=46.720, j4=-3.650, j5=80.274, j6=-5.969}
  [856] = {j1=-10.996, j2=63.563, j3=47.100, j4=-3.608, j5=79.971, j6=-6.368}
  [857] = {j1=-11.014, j2=63.114, j3=47.461, j4=-3.559, j5=79.696, j6=-6.753}
  [858] = {j1=-11.033, j2=62.671, j3=47.811, j4=-3.507, j5=79.442, j6=-7.126}
  [859] = {j1=-11.055, j2=62.230, j3=48.156, j4=-3.451, j5=79.200, j6=-7.492}
  [860] = {j1=-11.077, j2=61.787, j3=48.506, j4=-3.393, j5=78.962, j6=-7.855}
  [861] = {j1=-11.101, j2=61.337, j3=48.867, j4=-3.335, j5=78.720, j6=-8.219}
  [862] = {j1=-11.120, j2=60.935, j3=49.197, j4=-3.295, j5=78.499, j6=-8.533}
  [863] = {j1=-11.132, j2=60.531, j3=49.532, j4=-3.277, j5=78.277, j6=-8.831}
  [864] = {j1=-11.139, j2=60.130, j3=49.864, j4=-3.279, j5=78.065, j6=-9.108}
  [865] = {j1=-11.140, j2=59.737, j3=50.180, j4=-3.299, j5=77.873, j6=-9.360}
  [866] = {j1=-11.140, j2=59.721, j3=50.194, j4=-3.299, j5=77.863, j6=-9.368}
  [867] = {j1=-11.141, j2=59.755, j3=50.134, j4=-3.294, j5=77.950, j6=-9.312}
  [868] = {j1=-11.142, j2=59.767, j3=50.126, j4=-3.292, j5=77.952, j6=-9.304}
  [869] = {j1=-11.141, j2=60.156, j3=49.817, j4=-3.271, j5=78.135, j6=-9.052}
  [870] = {j1=-11.134, j2=60.553, j3=49.494, j4=-3.268, j5=78.339, j6=-8.775}
  [871] = {j1=-11.122, j2=60.953, j3=49.167, j4=-3.286, j5=78.551, j6=-8.477}
  [872] = {j1=-11.104, j2=61.349, j3=48.845, j4=-3.325, j5=78.762, j6=-8.164}
  [873] = {j1=-11.080, j2=61.794, j3=48.493, j4=-3.383, j5=78.994, j6=-7.801}
  [874] = {j1=-11.058, j2=62.233, j3=48.152, j4=-3.440, j5=79.222, j6=-7.439}
  [875] = {j1=-11.037, j2=62.669, j3=47.816, j4=-3.495, j5=79.453, j6=-7.074}
  [876] = {j1=-11.017, j2=63.107, j3=47.475, j4=-3.546, j5=79.697, j6=-6.702}
  [877] = {j1=-11.000, j2=63.551, j3=47.122, j4=-3.594, j5=79.962, j6=-6.319}
  [878] = {j1=-10.984, j2=64.006, j3=46.751, j4=-3.635, j5=80.255, j6=-5.921}
  [879] = {j1=-10.970, j2=64.474, j3=46.353, j4=-3.668, j5=80.585, j6=-5.505}
  [880] = {j1=-10.968, j2=64.556, j3=46.284, j4=-3.674, j5=80.643, j6=-5.430}
  [881] = {j1=-10.945, j2=65.033, j3=45.867, j4=-3.745, j5=81.002, j6=-4.975}
  [882] = {j1=-10.899, j2=65.574, j3=45.418, j4=-3.905, j5=81.376, j6=-4.424}
  [883] = {j1=-10.836, j2=66.049, j3=45.091, j4=-4.146, j5=81.601, j6=-3.918}
  [884] = {j1=-10.781, j2=66.365, j3=44.958, j4=-4.368, j5=81.620, j6=-3.590}
  [885] = {j1=-10.731, j2=66.618, j3=44.935, j4=-4.585, j5=81.499, j6=-3.350}
  [886] = {j1=-10.683, j2=66.821, j3=45.003, j4=-4.800, j5=81.263, j6=-3.184}
  [887] = {j1=-10.637, j2=66.982, j3=45.141, j4=-5.017, j5=80.934, j6=-3.075}
  [888] = {j1=-10.592, j2=67.111, j3=45.331, j4=-5.240, j5=80.533, j6=-3.009}
  [889] = {j1=-10.545, j2=67.218, j3=45.555, j4=-5.475, j5=80.084, j6=-2.970}
  [890] = {j1=-10.543, j2=67.259, j3=45.483, j4=-5.482, j5=80.216, j6=-2.871}
  [891] = {j1=-10.590, j2=67.149, j3=45.267, j4=-5.245, j5=80.654, j6=-2.913}
  [892] = {j1=-10.637, j2=67.015, j3=45.085, j4=-5.019, j5=81.041, j6=-2.982}
  [893] = {j1=-10.683, j2=66.849, j3=44.955, j4=-4.799, j5=81.359, j6=-3.094}
  [894] = {j1=-10.732, j2=66.642, j3=44.895, j4=-4.581, j5=81.583, j6=-3.264}
  [895] = {j1=-10.783, j2=66.383, j3=44.926, j4=-4.361, j5=81.692, j6=-3.507}
  [896] = {j1=-10.839, j2=66.063, j3=45.067, j4=-4.134, j5=81.663, j6=-3.839}
  [897] = {j1=-10.903, j2=65.585, j3=45.400, j4=-3.889, j5=81.429, j6=-4.347}
  [898] = {j1=-10.950, j2=65.041, j3=45.854, j4=-3.726, j5=81.049, j6=-4.898}
  [899] = {j1=-10.973, j2=64.561, j3=46.275, j4=-3.655, j5=80.684, j6=-5.352}
  [900] = {j1=-10.975, j2=64.476, j3=46.351, j4=-3.648, j5=80.617, j6=-5.427}
  [901] = {j1=-10.989, j2=64.005, j3=46.753, j4=-3.615, j5=80.281, j6=-5.841}
  [902] = {j1=-11.005, j2=63.548, j3=47.129, j4=-3.574, j5=79.982, j6=-6.237}
  [903] = {j1=-11.023, j2=63.101, j3=47.486, j4=-3.527, j5=79.711, j6=-6.619}
  [904] = {j1=-11.042, j2=62.660, j3=47.832, j4=-3.474, j5=79.462, j6=-6.990}
  [905] = {j1=-11.063, j2=62.221, j3=48.173, j4=-3.418, j5=79.224, j6=-7.353}
  [906] = {j1=-11.086, j2=61.780, j3=48.519, j4=-3.360, j5=78.991, j6=-7.714}
  [907] = {j1=-11.110, j2=61.332, j3=48.876, j4=-3.300, j5=78.752, j6=-8.077}
  [908] = {j1=-11.129, j2=60.932, j3=49.203, j4=-3.259, j5=78.534, j6=-8.389}
  [909] = {j1=-11.142, j2=60.530, j3=49.536, j4=-3.240, j5=78.315, j6=-8.686}
  [910] = {j1=-11.149, j2=60.129, j3=49.866, j4=-3.242, j5=78.104, j6=-8.963}
  [911] = {j1=-11.150, j2=59.736, j3=50.183, j4=-3.263, j5=77.911, j6=-9.215}
  [912] = {j1=-11.150, j2=59.719, j3=50.198, j4=-3.264, j5=77.900, j6=-9.224}
  [913] = {j1=-11.151, j2=59.755, j3=50.134, j4=-3.258, j5=77.991, j6=-9.165}
  [914] = {j1=-11.151, j2=59.767, j3=50.127, j4=-3.256, j5=77.993, j6=-9.156}
  [915] = {j1=-11.151, j2=60.156, j3=49.819, j4=-3.234, j5=78.176, j6=-8.905}
  [916] = {j1=-11.144, j2=60.552, j3=49.498, j4=-3.231, j5=78.377, j6=-8.628}
  [917] = {j1=-11.132, j2=60.949, j3=49.174, j4=-3.249, j5=78.586, j6=-8.332}
  [918] = {j1=-11.113, j2=61.344, j3=48.856, j4=-3.289, j5=78.793, j6=-8.020}
  [919] = {j1=-11.089, j2=61.786, j3=48.508, j4=-3.348, j5=79.021, j6=-7.658}
  [920] = {j1=-11.067, j2=62.222, j3=48.172, j4=-3.406, j5=79.243, j6=-7.298}
  [921] = {j1=-11.046, j2=62.656, j3=47.839, j4=-3.461, j5=79.470, j6=-6.935}
  [922] = {j1=-11.026, j2=63.092, j3=47.502, j4=-3.513, j5=79.709, j6=-6.566}
  [923] = {j1=-11.009, j2=63.534, j3=47.154, j4=-3.559, j5=79.969, j6=-6.185}
  [924] = {j1=-10.994, j2=63.986, j3=46.787, j4=-3.598, j5=80.258, j6=-5.790}
  [925] = {j1=-10.981, j2=64.452, j3=46.394, j4=-3.630, j5=80.584, j6=-5.377}
  [926] = {j1=-10.978, j2=64.533, j3=46.325, j4=-3.635, j5=80.641, j6=-5.302}
  [927] = {j1=-10.955, j2=65.009, j3=45.912, j4=-3.706, j5=80.996, j6=-4.849}
  [928] = {j1=-10.909, j2=65.547, j3=45.466, j4=-3.869, j5=81.366, j6=-4.298}
  [929] = {j1=-10.844, j2=66.022, j3=45.140, j4=-4.115, j5=81.592, j6=-3.788}
  [930] = {j1=-10.788, j2=66.339, j3=45.004, j4=-4.343, j5=81.613, j6=-3.454}
  [931] = {j1=-10.736, j2=66.595, j3=44.978, j4=-4.564, j5=81.497, j6=-3.209}
  [932] = {j1=-10.688, j2=66.800, j3=45.041, j4=-4.783, j5=81.267, j6=-3.036}
  [933] = {j1=-10.641, j2=66.965, j3=45.174, j4=-5.003, j5=80.945, j6=-2.921}
  [934] = {j1=-10.595, j2=67.097, j3=45.359, j4=-5.230, j5=80.552, j6=-2.848}
  [935] = {j1=-10.547, j2=67.206, j3=45.578, j4=-5.467, j5=80.110, j6=-2.804}
  [936] = {j1=-10.546, j2=67.232, j3=45.534, j4=-5.471, j5=80.191, j6=-2.741}
  [937] = {j1=-10.594, j2=67.118, j3=45.322, j4=-5.232, j5=80.622, j6=-2.787}
  [938] = {j1=-10.641, j2=66.981, j3=45.146, j4=-5.003, j5=81.004, j6=-2.862}
  [939] = {j1=-10.688, j2=66.812, j3=45.021, j4=-4.781, j5=81.314, j6=-2.979}
  [940] = {j1=-10.737, j2=66.602, j3=44.966, j4=-4.560, j5=81.533, j6=-3.155}
  [941] = {j1=-10.790, j2=66.342, j3=45.001, j4=-4.336, j5=81.638, j6=-3.402}
  [942] = {j1=-10.847, j2=66.020, j3=45.144, j4=-4.104, j5=81.606, j6=-3.737}
  [943] = {j1=-10.912, j2=65.541, j3=45.478, j4=-3.856, j5=81.372, j6=-4.249}
  [944] = {j1=-10.959, j2=64.999, j3=45.930, j4=-3.691, j5=80.993, j6=-4.800}
  [945] = {j1=-10.983, j2=64.520, j3=46.349, j4=-3.619, j5=80.631, j6=-5.252}
  [946] = {j1=-10.985, j2=64.435, j3=46.425, j4=-3.613, j5=80.564, j6=-5.327}
  [947] = {j1=-10.998, j2=63.965, j3=46.824, j4=-3.581, j5=80.231, j6=-5.739}
  [948] = {j1=-11.014, j2=63.509, j3=47.198, j4=-3.541, j5=79.934, j6=-6.133}
  [949] = {j1=-11.032, j2=63.064, j3=47.553, j4=-3.494, j5=79.666, j6=-6.513}
  [950] = {j1=-11.051, j2=62.624, j3=47.897, j4=-3.442, j5=79.418, j6=-6.882}
  [951] = {j1=-11.072, j2=62.186, j3=48.237, j4=-3.386, j5=79.183, j6=-7.244}
  [952] = {j1=-11.095, j2=61.746, j3=48.580, j4=-3.327, j5=78.952, j6=-7.604}
  [953] = {j1=-11.120, j2=61.299, j3=48.936, j4=-3.266, j5=78.716, j6=-7.966}
  [954] = {j1=-11.139, j2=60.901, j3=49.260, j4=-3.224, j5=78.500, j6=-8.278}
  [955] = {j1=-11.152, j2=60.499, j3=49.592, j4=-3.205, j5=78.283, j6=-8.574}
  [956] = {j1=-11.159, j2=60.099, j3=49.921, j4=-3.207, j5=78.073, j6=-8.850}
  [957] = {j1=-11.160, j2=59.705, j3=50.238, j4=-3.229, j5=77.879, j6=-9.101}
  [958] = {j1=-11.160, j2=59.689, j3=50.253, j4=-3.229, j5=77.868, j6=-9.110}
  [959] = {j1=-11.161, j2=59.725, j3=50.189, j4=-3.223, j5=77.959, j6=-9.051}
  [960] = {j1=-11.161, j2=59.736, j3=50.183, j4=-3.221, j5=77.960, j6=-9.042}
  [961] = {j1=-11.161, j2=60.124, j3=49.875, j4=-3.199, j5=78.143, j6=-8.791}
  [962] = {j1=-11.154, j2=60.519, j3=49.556, j4=-3.195, j5=78.341, j6=-8.516}
  [963] = {j1=-11.142, j2=60.915, j3=49.235, j4=-3.214, j5=78.547, j6=-8.221}
  [964] = {j1=-11.123, j2=61.308, j3=48.920, j4=-3.255, j5=78.751, j6=-7.910}
  [965] = {j1=-11.099, j2=61.749, j3=48.575, j4=-3.315, j5=78.975, j6=-7.549}
  [966] = {j1=-11.076, j2=62.184, j3=48.241, j4=-3.373, j5=79.195, j6=-7.189}
  [967] = {j1=-11.055, j2=62.616, j3=47.911, j4=-3.429, j5=79.419, j6=-6.827}
  [968] = {j1=-11.036, j2=63.051, j3=47.576, j4=-3.480, j5=79.656, j6=-6.459}
  [969] = {j1=-11.018, j2=63.492, j3=47.230, j4=-3.525, j5=79.913, j6=-6.080}
  [970] = {j1=-11.003, j2=63.942, j3=46.865, j4=-3.564, j5=80.199, j6=-5.687}
  [971] = {j1=-10.990, j2=64.407, j3=46.475, j4=-3.594, j5=80.521, j6=-5.276}
  [972] = {j1=-10.988, j2=64.487, j3=46.407, j4=-3.599, j5=80.577, j6=-5.202}
  [973] = {j1=-10.965, j2=64.961, j3=45.997, j4=-3.669, j5=80.928, j6=-4.751}
  [974] = {j1=-10.918, j2=65.498, j3=45.554, j4=-3.834, j5=81.296, j6=-4.199}
  [975] = {j1=-10.852, j2=65.973, j3=45.229, j4=-4.084, j5=81.520, j6=-3.687}
  [976] = {j1=-10.795, j2=66.291, j3=45.091, j4=-4.316, j5=81.543, j6=-3.350}
  [977] = {j1=-10.742, j2=66.549, j3=45.062, j4=-4.541, j5=81.431, j6=-3.099}
  [978] = {j1=-10.693, j2=66.756, j3=45.121, j4=-4.763, j5=81.205, j6=-2.921}
  [979] = {j1=-10.645, j2=66.923, j3=45.249, j4=-4.986, j5=80.889, j6=-2.801}
  [980] = {j1=-10.599, j2=67.059, j3=45.429, j4=-5.215, j5=80.502, j6=-2.723}
  [981] = {j1=-10.551, j2=67.170, j3=45.643, j4=-5.454, j5=80.065, j6=-2.674}
  [982] = {j1=-10.550, j2=67.195, j3=45.600, j4=-5.457, j5=80.146, j6=-2.612}
  [983] = {j1=-10.598, j2=67.079, j3=45.394, j4=-5.217, j5=80.571, j6=-2.662}
  [984] = {j1=-10.645, j2=66.939, j3=45.223, j4=-4.986, j5=80.945, j6=-2.742}
  [985] = {j1=-10.694, j2=66.766, j3=45.104, j4=-4.760, j5=81.249, j6=-2.865}
  [986] = {j1=-10.744, j2=66.553, j3=45.054, j4=-4.536, j5=81.461, j6=-3.045}
  [987] = {j1=-10.797, j2=66.290, j3=45.092, j4=-4.309, j5=81.562, j6=-3.297}
  [988] = {j1=-10.855, j2=65.968, j3=45.238, j4=-4.073, j5=81.528, j6=-3.637}
  [989] = {j1=-10.922, j2=65.489, j3=45.571, j4=-3.820, j5=81.294, j6=-4.150}
  [990] = {j1=-10.970, j2=64.948, j3=46.021, j4=-3.653, j5=80.919, j6=-4.701}
  [991] = {j1=-10.993, j2=64.470, j3=46.437, j4=-3.582, j5=80.559, j6=-5.151}
  [992] = {j1=-10.995, j2=64.385, j3=46.513, j4=-3.576, j5=80.493, j6=-5.225}
  [993] = {j1=-11.008, j2=63.917, j3=46.911, j4=-3.545, j5=80.162, j6=-5.635}
  [994] = {j1=-11.024, j2=63.462, j3=47.283, j4=-3.506, j5=79.867, j6=-6.027}
  [995] = {j1=-11.041, j2=63.017, j3=47.637, j4=-3.460, j5=79.600, j6=-6.406}
  [996] = {j1=-11.061, j2=62.578, j3=47.980, j4=-3.408, j5=79.353, j6=-6.774}
  [997] = {j1=-11.082, j2=62.140, j3=48.319, j4=-3.351, j5=79.119, j6=-7.136}
  [998] = {j1=-11.105, j2=61.701, j3=48.661, j4=-3.291, j5=78.889, j6=-7.495}
  [999] = {j1=-11.130, j2=61.255, j3=49.015, j4=-3.230, j5=78.656, j6=-7.856}
  [1000] = {j1=-11.150, j2=60.858, j3=49.338, j4=-3.187, j5=78.442, j6=-8.167}
  [1001] = {j1=-11.163, j2=60.457, j3=49.667, j4=-3.167, j5=78.227, j6=-8.462}
  [1002] = {j1=-11.170, j2=60.058, j3=49.995, j4=-3.169, j5=78.019, j6=-8.737}
  [1003] = {j1=-11.170, j2=59.664, j3=50.311, j4=-3.191, j5=77.826, j6=-8.988}
  [1004] = {j1=-11.171, j2=59.648, j3=50.327, j4=-3.192, j5=77.814, j6=-8.997}
  [1005] = {j1=-11.171, j2=59.683, j3=50.264, j4=-3.186, j5=77.904, j6=-8.937}
  [1006] = {j1=-11.172, j2=59.695, j3=50.258, j4=-3.184, j5=77.905, j6=-8.929}
  [1007] = {j1=-11.172, j2=60.082, j3=49.952, j4=-3.161, j5=78.086, j6=-8.679}
  [1008] = {j1=-11.165, j2=60.475, j3=49.635, j4=-3.157, j5=78.282, j6=-8.405}
  [1009] = {j1=-11.152, j2=60.870, j3=49.317, j4=-3.176, j5=78.484, j6=-8.111}
  [1010] = {j1=-11.133, j2=61.261, j3=49.005, j4=-3.218, j5=78.684, j6=-7.801}
  [1011] = {j1=-11.109, j2=61.701, j3=48.662, j4=-3.279, j5=78.906, j6=-7.440}
  [1012] = {j1=-11.086, j2=62.134, j3=48.330, j4=-3.338, j5=79.123, j6=-7.081}
  [1013] = {j1=-11.065, j2=62.566, j3=48.001, j4=-3.393, j5=79.346, j6=-6.720}
  [1014] = {j1=-11.045, j2=63.000, j3=47.668, j4=-3.444, j5=79.581, j6=-6.352}
  [1015] = {j1=-11.028, j2=63.440, j3=47.323, j4=-3.489, j5=79.836, j6=-5.974}
  [1016] = {j1=-11.013, j2=63.889, j3=46.961, j4=-3.526, j5=80.119, j6=-5.582}
  [1017] = {j1=-11.001, j2=64.352, j3=46.573, j4=-3.555, j5=80.438, j6=-5.174}
  [1018] = {j1=-10.999, j2=64.432, j3=46.506, j4=-3.560, j5=80.493, j6=-5.100}
  [1019] = {j1=-10.976, j2=64.904, j3=46.100, j4=-3.629, j5=80.839, j6=-4.651}
  [1020] = {j1=-10.928, j2=65.439, j3=45.660, j4=-3.796, j5=81.202, j6=-4.101}
  [1021] = {j1=-10.861, j2=65.913, j3=45.336, j4=-4.050, j5=81.425, j6=-3.586}
  [1022] = {j1=-10.803, j2=66.232, j3=45.197, j4=-4.287, j5=81.449, j6=-3.245}
  [1023] = {j1=-10.749, j2=66.491, j3=45.165, j4=-4.515, j5=81.340, j6=-2.990}
  [1024] = {j1=-10.699, j2=66.702, j3=45.219, j4=-4.740, j5=81.119, j6=-2.807}
  [1025] = {j1=-10.651, j2=66.872, j3=45.342, j4=-4.966, j5=80.809, j6=-2.681}
  [1026] = {j1=-10.603, j2=67.010, j3=45.516, j4=-5.197, j5=80.428, j6=-2.598}
  [1027] = {j1=-10.555, j2=67.125, j3=45.726, j4=-5.438, j5=79.997, j6=-2.544}
  [1028] = {j1=-10.554, j2=67.149, j3=45.683, j4=-5.442, j5=80.077, j6=-2.482}
  [1029] = {j1=-10.603, j2=67.029, j3=45.483, j4=-5.199, j5=80.494, j6=-2.537}
  [1030] = {j1=-10.651, j2=66.885, j3=45.318, j4=-4.966, j5=80.861, j6=-2.623}
  [1031] = {j1=-10.700, j2=66.710, j3=45.205, j4=-4.737, j5=81.158, j6=-2.751}
  [1032] = {j1=-10.751, j2=66.494, j3=45.161, j4=-4.510, j5=81.365, j6=-2.936}
  [1033] = {j1=-10.805, j2=66.228, j3=45.203, j4=-4.279, j5=81.461, j6=-3.193}
  [1034] = {j1=-10.865, j2=65.904, j3=45.351, j4=-4.039, j5=81.425, j6=-3.536}
  [1035] = {j1=-10.932, j2=65.426, j3=45.684, j4=-3.781, j5=81.193, j6=-4.051}
  [1036] = {j1=-10.981, j2=64.887, j3=46.130, j4=-3.612, j5=80.821, j6=-4.601}
  [1037] = {j1=-11.004, j2=64.411, j3=46.544, j4=-3.542, j5=80.465, j6=-5.049}
  [1038] = {j1=-11.006, j2=64.326, j3=46.620, j4=-3.536, j5=80.399, j6=-5.122}
  [1039] = {j1=-11.019, j2=63.858, j3=47.016, j4=-3.507, j5=80.070, j6=-5.530}
  [1040] = {j1=-11.034, j2=63.404, j3=47.387, j4=-3.468, j5=79.776, j6=-5.921}
  [1041] = {j1=-11.051, j2=62.959, j3=47.741, j4=-3.423, j5=79.509, j6=-6.298}
  [1042] = {j1=-11.071, j2=62.520, j3=48.084, j4=-3.371, j5=79.263, j6=-6.667}
  [1043] = {j1=-11.093, j2=62.083, j3=48.423, j4=-3.314, j5=79.029, j6=-7.028}
  [1044] = {j1=-11.116, j2=61.643, j3=48.764, j4=-3.253, j5=78.800, j6=-7.388}
  [1045] = {j1=-11.142, j2=61.198, j3=49.117, j4=-3.190, j5=78.568, j6=-7.748}
  [1046] = {j1=-11.161, j2=60.802, j3=49.438, j4=-3.147, j5=78.357, j6=-8.058}
  [1047] = {j1=-11.175, j2=60.402, j3=49.766, j4=-3.127, j5=78.144, j6=-8.352}
  [1048] = {j1=-11.181, j2=60.004, j3=50.092, j4=-3.129, j5=77.937, j6=-8.625}
  [1049] = {j1=-11.182, j2=59.611, j3=50.408, j4=-3.151, j5=77.745, j6=-8.875}
  [1050] = {j1=-11.182, j2=59.594, j3=50.424, j4=-3.152, j5=77.732, j6=-8.884}
  [1051] = {j1=-11.183, j2=59.629, j3=50.362, j4=-3.146, j5=77.822, j6=-8.824}
  [1052] = {j1=-11.184, j2=59.640, j3=50.356, j4=-3.144, j5=77.822, j6=-8.816}
  [1053] = {j1=-11.183, j2=60.026, j3=50.052, j4=-3.120, j5=78.001, j6=-8.567}
  [1054] = {j1=-11.177, j2=60.418, j3=49.738, j4=-3.116, j5=78.193, j6=-8.295}
  [1055] = {j1=-11.164, j2=60.811, j3=49.423, j4=-3.135, j5=78.392, j6=-8.002}
  [1056] = {j1=-11.145, j2=61.200, j3=49.114, j4=-3.178, j5=78.589, j6=-7.693}
  [1057] = {j1=-11.120, j2=61.639, j3=48.773, j4=-3.240, j5=78.807, j6=-7.333}
  [1058] = {j1=-11.097, j2=62.072, j3=48.442, j4=-3.299, j5=79.024, j6=-6.974}
  [1059] = {j1=-11.075, j2=62.503, j3=48.113, j4=-3.355, j5=79.245, j6=-6.612}
  [1060] = {j1=-11.056, j2=62.937, j3=47.781, j4=-3.405, j5=79.479, j6=-6.244}
  [1061] = {j1=-11.039, j2=63.376, j3=47.437, j4=-3.450, j5=79.733, j6=-5.867}
  [1062] = {j1=-11.024, j2=63.824, j3=47.076, j4=-3.486, j5=80.014, j6=-5.477}
  [1063] = {j1=-11.012, j2=64.285, j3=46.692, j4=-3.513, j5=80.329, j6=-5.071}
  [1064] = {j1=-11.010, j2=64.365, j3=46.626, j4=-3.518, j5=80.383, j6=-4.997}
  [1065] = {j1=-10.988, j2=64.834, j3=46.223, j4=-3.587, j5=80.724, j6=-4.551}
  [1066] = {j1=-10.939, j2=65.367, j3=45.788, j4=-3.755, j5=81.082, j6=-4.002}
  [1067] = {j1=-10.871, j2=65.840, j3=45.465, j4=-4.014, j5=81.301, j6=-3.486}
  [1068] = {j1=-10.812, j2=66.160, j3=45.326, j4=-4.255, j5=81.326, j6=-3.141}
  [1069] = {j1=-10.757, j2=66.421, j3=45.290, j4=-4.487, j5=81.220, j6=-2.882}
  [1070] = {j1=-10.706, j2=66.634, j3=45.340, j4=-4.715, j5=81.004, j6=-2.693}
  [1071] = {j1=-10.657, j2=66.808, j3=45.457, j4=-4.943, j5=80.699, j6=-2.562}
  [1072] = {j1=-10.609, j2=66.949, j3=45.626, j4=-5.176, j5=80.325, j6=-2.473}
  [1073] = {j1=-10.560, j2=67.067, j3=45.830, j4=-5.419, j5=79.900, j6=-2.414}
  [1074] = {j1=-10.559, j2=67.092, j3=45.787, j4=-5.423, j5=79.980, j6=-2.352}
  [1075] = {j1=-10.608, j2=66.968, j3=45.594, j4=-5.178, j5=80.389, j6=-2.413}
  [1076] = {j1=-10.657, j2=66.820, j3=45.436, j4=-4.942, j5=80.748, j6=-2.504}
  [1077] = {j1=-10.707, j2=66.640, j3=45.330, j4=-4.711, j5=81.038, j6=-2.638}
  [1078] = {j1=-10.759, j2=66.421, j3=45.292, j4=-4.480, j5=81.238, j6=-2.828}
  [1079] = {j1=-10.814, j2=66.153, j3=45.338, j4=-4.245, j5=81.330, j6=-3.089}
  [1080] = {j1=-10.875, j2=65.828, j3=45.488, j4=-4.001, j5=81.293, j6=-3.435}
  [1081] = {j1=-10.944, j2=65.350, j3=45.819, j4=-3.739, j5=81.062, j6=-3.952}
  [1082] = {j1=-10.992, j2=64.813, j3=46.263, j4=-3.569, j5=80.695, j6=-4.500}
  [1083] = {j1=-11.016, j2=64.338, j3=46.673, j4=-3.498, j5=80.343, j6=-4.945}
  [1084] = {j1=-11.018, j2=64.253, j3=46.749, j4=-3.493, j5=80.276, j6=-5.018}
  [1085] = {j1=-11.030, j2=63.787, j3=47.144, j4=-3.465, j5=79.950, j6=-5.424}
  [1086] = {j1=-11.045, j2=63.333, j3=47.515, j4=-3.427, j5=79.656, j6=-5.814}
  [1087] = {j1=-11.063, j2=62.887, j3=47.869, j4=-3.382, j5=79.389, j6=-6.191}
  [1088] = {j1=-11.083, j2=62.448, j3=48.213, j4=-3.330, j5=79.142, j6=-6.559}
  [1089] = {j1=-11.104, j2=62.010, j3=48.553, j4=-3.273, j5=78.907, j6=-6.922}
  [1090] = {j1=-11.128, j2=61.570, j3=48.895, j4=-3.212, j5=78.678, j6=-7.281}
  [1091] = {j1=-11.154, j2=61.126, j3=49.247, j4=-3.148, j5=78.446, j6=-7.642}
  [1092] = {j1=-11.174, j2=60.730, j3=49.567, j4=-3.103, j5=78.237, j6=-7.951}
  [1093] = {j1=-11.187, j2=60.331, j3=49.893, j4=-3.082, j5=78.027, j6=-8.243}
  [1094] = {j1=-11.194, j2=59.934, j3=50.217, j4=-3.084, j5=77.822, j6=-8.514}
  [1095] = {j1=-11.195, j2=59.541, j3=50.532, j4=-3.107, j5=77.631, j6=-8.763}
  [1096] = {j1=-11.195, j2=59.524, j3=50.549, j4=-3.108, j5=77.618, j6=-8.772}
  [1097] = {j1=-11.196, j2=59.559, j3=50.487, j4=-3.102, j5=77.707, j6=-8.712}
  [1098] = {j1=-11.197, j2=59.569, j3=50.482, j4=-3.100, j5=77.706, j6=-8.703}
  [1099] = {j1=-11.197, j2=59.954, j3=50.181, j4=-3.075, j5=77.882, j6=-8.456}
  [1100] = {j1=-11.190, j2=60.344, j3=49.870, j4=-3.071, j5=78.070, j6=-8.186}
  [1101] = {j1=-11.177, j2=60.735, j3=49.558, j4=-3.091, j5=78.264, j6=-7.895}
  [1102] = {j1=-11.158, j2=61.123, j3=49.252, j4=-3.134, j5=78.458, j6=-7.587}
  [1103] = {j1=-11.132, j2=61.561, j3=48.912, j4=-3.197, j5=78.674, j6=-7.227}
  [1104] = {j1=-11.109, j2=61.994, j3=48.582, j4=-3.257, j5=78.889, j6=-6.867}
  [1105] = {j1=-11.087, j2=62.425, j3=48.253, j4=-3.313, j5=79.110, j6=-6.505}
  [1106] = {j1=-11.068, j2=62.859, j3=47.921, j4=-3.363, j5=79.344, j6=-6.137}
  [1107] = {j1=-11.051, j2=63.297, j3=47.578, j4=-3.407, j5=79.597, j6=-5.759}
  [1108] = {j1=-11.037, j2=63.745, j3=47.218, j4=-3.442, j5=79.876, j6=-5.370}
  [1109] = {j1=-11.025, j2=64.205, j3=46.836, j4=-3.468, j5=80.188, j6=-4.966}
  [1110] = {j1=-11.023, j2=64.284, j3=46.771, j4=-3.472, j5=80.240, j6=-4.894}
  [1111] = {j1=-11.000, j2=64.751, j3=46.373, j4=-3.541, j5=80.577, j6=-4.450}
  [1112] = {j1=-10.951, j2=65.281, j3=45.942, j4=-3.711, j5=80.927, j6=-3.903}
  [1113] = {j1=-10.882, j2=65.752, j3=45.622, j4=-3.974, j5=81.143, j6=-3.386}
  [1114] = {j1=-10.821, j2=66.072, j3=45.481, j4=-4.218, j5=81.167, j6=-3.038}
  [1115] = {j1=-10.766, j2=66.336, j3=45.442, j4=-4.454, j5=81.064, j6=-2.774}
  [1116] = {j1=-10.714, j2=66.552, j3=45.487, j4=-4.685, j5=80.853, j6=-2.580}
  [1117] = {j1=-10.664, j2=66.728, j3=45.599, j4=-4.916, j5=80.554, j6=-2.443}
  [1118] = {j1=-10.615, j2=66.874, j3=45.761, j4=-5.152, j5=80.186, j6=-2.348}
  [1119] = {j1=-10.566, j2=66.996, j3=45.959, j4=-5.397, j5=79.768, j6=-2.284}
  [1120] = {j1=-10.565, j2=67.019, j3=45.917, j4=-5.400, j5=79.847, j6=-2.221}
  [1121] = {j1=-10.615, j2=66.891, j3=45.731, j4=-5.153, j5=80.248, j6=-2.288}
  [1122] = {j1=-10.664, j2=66.739, j3=45.581, j4=-4.915, j5=80.599, j6=-2.385}
  [1123] = {j1=-10.715, j2=66.555, j3=45.482, j4=-4.681, j5=80.881, j6=-2.524}
  [1124] = {j1=-10.768, j2=66.332, j3=45.450, j4=-4.447, j5=81.075, j6=-2.720}
  [1125] = {j1=-10.824, j2=66.061, j3=45.501, j4=-4.208, j5=81.162, j6=-2.986}
  [1126] = {j1=-10.886, j2=65.735, j3=45.653, j4=-3.960, j5=81.124, j6=-3.335}
  [1127] = {j1=-10.956, j2=65.258, j3=45.983, j4=-3.694, j5=80.896, j6=-3.852}
  [1128] = {j1=-11.005, j2=64.723, j3=46.423, j4=-3.521, j5=80.534, j6=-4.398}
  [1129] = {j1=-11.029, j2=64.250, j3=46.831, j4=-3.451, j5=80.186, j6=-4.840}
  [1130] = {j1=-11.031, j2=64.165, j3=46.907, j4=-3.445, j5=80.119, j6=-4.913}
  [1131] = {j1=-11.043, j2=63.699, j3=47.300, j4=-3.419, j5=79.794, j6=-5.316}
  [1132] = {j1=-11.058, j2=63.245, j3=47.672, j4=-3.382, j5=79.500, j6=-5.705}
  [1133] = {j1=-11.076, j2=62.799, j3=48.028, j4=-3.337, j5=79.232, j6=-6.083}
  [1134] = {j1=-11.095, j2=62.358, j3=48.374, j4=-3.285, j5=78.982, j6=-6.452}
  [1135] = {j1=-11.118, j2=61.919, j3=48.716, j4=-3.227, j5=78.745, j6=-6.815}
  [1136] = {j1=-11.142, j2=61.479, j3=49.059, j4=-3.165, j5=78.515, j6=-7.176}
  [1137] = {j1=-11.168, j2=61.034, j3=49.412, j4=-3.100, j5=78.284, j6=-7.536}
  [1138] = {j1=-11.188, j2=60.639, j3=49.730, j4=-3.055, j5=78.076, j6=-7.845}
  [1139] = {j1=-11.202, j2=60.241, j3=50.054, j4=-3.034, j5=77.868, j6=-8.135}
  [1140] = {j1=-11.209, j2=59.844, j3=50.377, j4=-3.035, j5=77.666, j6=-8.405}
  [1141] = {j1=-11.209, j2=59.452, j3=50.691, j4=-3.059, j5=77.477, j6=-8.651}
  [1142] = {j1=-11.210, j2=59.435, j3=50.709, j4=-3.059, j5=77.462, j6=-8.660}
  [1143] = {j1=-11.211, j2=59.469, j3=50.647, j4=-3.053, j5=77.552, j6=-8.599}
  [1144] = {j1=-11.211, j2=59.480, j3=50.643, j4=-3.051, j5=77.550, j6=-8.591}
  [1145] = {j1=-11.211, j2=59.863, j3=50.344, j4=-3.026, j5=77.721, j6=-8.346}
  [1146] = {j1=-11.205, j2=60.250, j3=50.038, j4=-3.022, j5=77.905, j6=-8.078}
  [1147] = {j1=-11.192, j2=60.639, j3=49.730, j4=-3.041, j5=78.094, j6=-7.789}
  [1148] = {j1=-11.172, j2=61.026, j3=49.426, j4=-3.085, j5=78.284, j6=-7.482}
  [1149] = {j1=-11.146, j2=61.463, j3=49.088, j4=-3.149, j5=78.498, j6=-7.122}
  [1150] = {j1=-11.122, j2=61.896, j3=48.757, j4=-3.210, j5=78.713, j6=-6.761}
  [1151] = {j1=-11.101, j2=62.328, j3=48.428, j4=-3.266, j5=78.934, j6=-6.397}
  [1152] = {j1=-11.081, j2=62.762, j3=48.094, j4=-3.316, j5=79.169, j6=-6.028}
  [1153] = {j1=-11.064, j2=63.201, j3=47.750, j4=-3.359, j5=79.422, j6=-5.650}
  [1154] = {j1=-11.050, j2=63.648, j3=47.391, j4=-3.394, j5=79.700, j6=-5.262}
  [1155] = {j1=-11.039, j2=64.106, j3=47.012, j4=-3.418, j5=80.008, j6=-4.860}
  [1156] = {j1=-11.037, j2=64.184, j3=46.949, j4=-3.422, j5=80.058, j6=-4.788}
  [1157] = {j1=-11.014, j2=64.648, j3=46.555, j4=-3.490, j5=80.388, j6=-4.347}
  [1158] = {j1=-10.965, j2=65.175, j3=46.130, j4=-3.662, j5=80.731, j6=-3.803}
  [1159] = {j1=-10.894, j2=65.645, j3=45.813, j4=-3.929, j5=80.941, j6=-3.285}
  [1160] = {j1=-10.832, j2=65.966, j3=45.672, j4=-4.177, j5=80.965, j6=-2.934}
  [1161] = {j1=-10.776, j2=66.231, j3=45.629, j4=-4.416, j5=80.864, j6=-2.666}
  [1162] = {j1=-10.723, j2=66.450, j3=45.669, j4=-4.651, j5=80.658, j6=-2.467}
  [1163] = {j1=-10.673, j2=66.630, j3=45.774, j4=-4.884, j5=80.365, j6=-2.323}
  [1164] = {j1=-10.623, j2=66.780, j3=45.929, j4=-5.122, j5=80.004, j6=-2.223}
  [1165] = {j1=-10.573, j2=66.905, j3=46.121, j4=-5.369, j5=79.592, j6=-2.152}
  [1166] = {j1=-10.573, j2=66.929, j3=46.080, j4=-5.372, j5=79.669, j6=-2.090}
  [1167] = {j1=-10.623, j2=66.795, j3=45.903, j4=-5.123, j5=80.062, j6=-2.162}
  [1168] = {j1=-10.673, j2=66.638, j3=45.761, j4=-4.882, j5=80.403, j6=-2.265}
  [1169] = {j1=-10.724, j2=66.449, j3=45.671, j4=-4.646, j5=80.677, j6=-2.411}
  [1170] = {j1=-10.778, j2=66.222, j3=45.645, j4=-4.408, j5=80.864, j6=-2.612}
  [1171] = {j1=-10.836, j2=65.949, j3=45.702, j4=-4.166, j5=80.947, j6=-2.882}
  [1172] = {j1=-10.898, j2=65.621, j3=45.856, j4=-3.913, j5=80.907, j6=-3.234}
  [1173] = {j1=-10.970, j2=65.145, j3=46.184, j4=-3.643, j5=80.682, j6=-3.752}
  [1174] = {j1=-11.020, j2=64.612, j3=46.620, j4=-3.468, j5=80.326, j6=-4.295}
  [1175] = {j1=-11.043, j2=64.141, j3=47.025, j4=-3.398, j5=79.982, j6=-4.734}
  [1176] = {j1=-11.046, j2=64.056, j3=47.102, j4=-3.393, j5=79.915, j6=-4.807}
  [1177] = {j1=-11.057, j2=63.590, j3=47.494, j4=-3.367, j5=79.591, j6=-5.207}
  [1178] = {j1=-11.072, j2=63.135, j3=47.867, j4=-3.331, j5=79.296, j6=-5.596}
  [1179] = {j1=-11.090, j2=62.688, j3=48.226, j4=-3.286, j5=79.025, j6=-5.974}
  [1180] = {j1=-11.110, j2=62.245, j3=48.576, j4=-3.234, j5=78.772, j6=-6.345}
  [1181] = {j1=-11.133, j2=61.804, j3=48.921, j4=-3.176, j5=78.532, j6=-6.710}
  [1182] = {j1=-11.157, j2=61.362, j3=49.268, j4=-3.113, j5=78.298, j6=-7.072}
  [1183] = {j1=-11.184, j2=60.917, j3=49.621, j4=-3.047, j5=78.067, j6=-7.433}
  [1184] = {j1=-11.204, j2=60.522, j3=49.939, j4=-3.001, j5=77.860, j6=-7.740}
  [1185] = {j1=-11.218, j2=60.125, j3=50.262, j4=-2.979, j5=77.655, j6=-8.029}
  [1186] = {j1=-11.225, j2=59.730, j3=50.582, j4=-2.981, j5=77.456, j6=-8.296}
  [1187] = {j1=-11.226, j2=59.338, j3=50.896, j4=-3.004, j5=77.268, j6=-8.540}
  [1188] = {j1=-11.226, j2=59.320, j3=50.915, j4=-3.004, j5=77.252, j6=-8.549}
  [1189] = {j1=-11.227, j2=59.354, j3=50.854, j4=-2.998, j5=77.340, j6=-8.488}
  [1190] = {j1=-11.228, j2=59.363, j3=50.852, j4=-2.996, j5=77.337, j6=-8.480}
  [1191] = {j1=-11.228, j2=59.744, j3=50.557, j4=-2.970, j5=77.503, j6=-8.238}
  [1192] = {j1=-11.222, j2=60.130, j3=50.254, j4=-2.966, j5=77.681, j6=-7.972}
  [1193] = {j1=-11.208, j2=60.516, j3=49.950, j4=-2.986, j5=77.865, j6=-7.685}
  [1194] = {j1=-11.188, j2=60.901, j3=49.649, j4=-3.031, j5=78.051, j6=-7.379}
  [1195] = {j1=-11.162, j2=61.338, j3=49.312, j4=-3.095, j5=78.263, j6=-7.019}
  [1196] = {j1=-11.138, j2=61.771, j3=48.980, j4=-3.156, j5=78.478, j6=-6.656}
  [1197] = {j1=-11.116, j2=62.204, j3=48.649, j4=-3.212, j5=78.700, j6=-6.291}
  [1198] = {j1=-11.097, j2=62.639, j3=48.313, j4=-3.262, j5=78.936, j6=-5.920}
  [1199] = {j1=-11.080, j2=63.078, j3=47.969, j4=-3.305, j5=79.189, j6=-5.541}
  [1200] = {j1=-11.065, j2=63.525, j3=47.610, j4=-3.339, j5=79.466, j6=-5.153}
  [1201] = {j1=-11.054, j2=63.982, j3=47.233, j4=-3.362, j5=79.770, j6=-4.754}
  [1202] = {j1=-11.052, j2=64.059, j3=47.172, j4=-3.365, j5=79.818, j6=-4.682}
  [1203] = {j1=-11.030, j2=64.520, j3=46.783, j4=-3.433, j5=80.141, j6=-4.245}
  [1204] = {j1=-10.980, j2=65.044, j3=46.364, j4=-3.606, j5=80.475, j6=-3.703}
  [1205] = {j1=-10.908, j2=65.511, j3=46.051, j4=-3.877, j5=80.679, j6=-3.185}
  [1206] = {j1=-10.845, j2=65.832, j3=45.909, j4=-4.130, j5=80.701, j6=-2.831}
  [1207] = {j1=-10.788, j2=66.100, j3=45.863, j4=-4.372, j5=80.602, j6=-2.559}
  [1208] = {j1=-10.734, j2=66.322, j3=45.897, j4=-4.610, j5=80.400, j6=-2.354}
  [1209] = {j1=-10.683, j2=66.506, j3=45.996, j4=-4.846, j5=80.113, j6=-2.204}
  [1210] = {j1=-10.633, j2=66.660, j3=46.144, j4=-5.086, j5=79.759, j6=-2.097}
  [1211] = {j1=-10.582, j2=66.790, j3=46.327, j4=-5.336, j5=79.354, j6=-2.020}
  [1212] = {j1=-10.582, j2=66.813, j3=46.288, j4=-5.338, j5=79.429, j6=-1.958}
  [1213] = {j1=-10.633, j2=66.674, j3=46.121, j4=-5.087, j5=79.811, j6=-2.037}
  [1214] = {j1=-10.684, j2=66.510, j3=45.990, j4=-4.843, j5=80.143, j6=-2.146}
  [1215] = {j1=-10.736, j2=66.316, j3=45.908, j4=-4.603, j5=80.407, j6=-2.299}
  [1216] = {j1=-10.790, j2=66.084, j3=45.891, j4=-4.362, j5=80.587, j6=-2.505}
  [1217] = {j1=-10.849, j2=65.808, j3=45.953, j4=-4.116, j5=80.665, j6=-2.780}
  [1218] = {j1=-10.913, j2=65.478, j3=46.110, j4=-3.859, j5=80.623, j6=-3.135}
  [1219] = {j1=-10.986, j2=65.003, j3=46.438, j4=-3.585, j5=80.402, j6=-3.652}
  [1220] = {j1=-11.036, j2=64.472, j3=46.870, j4=-3.408, j5=80.052, j6=-4.193}
  [1221] = {j1=-11.060, j2=64.003, j3=47.272, j4=-3.338, j5=79.712, j6=-4.628}
  [1222] = {j1=-11.062, j2=63.917, j3=47.350, j4=-3.333, j5=79.644, j6=-4.700}
  [1223] = {j1=-11.074, j2=63.451, j3=47.743, j4=-3.308, j5=79.320, j6=-5.099}
  [1224] = {j1=-11.089, j2=62.995, j3=48.119, j4=-3.272, j5=79.023, j6=-5.487}
  [1225] = {j1=-11.107, j2=62.545, j3=48.482, j4=-3.228, j5=78.747, j6=-5.867}
  [1226] = {j1=-11.127, j2=62.099, j3=48.836, j4=-3.175, j5=78.489, j6=-6.240}
  [1227] = {j1=-11.150, j2=61.655, j3=49.187, j4=-3.117, j5=78.244, j6=-6.607}
  [1228] = {j1=-11.175, j2=61.211, j3=49.538, j4=-3.053, j5=78.007, j6=-6.971}
  [1229] = {j1=-11.202, j2=60.764, j3=49.894, j4=-2.985, j5=77.773, j6=-7.333}
  [1230] = {j1=-11.223, j2=60.369, j3=50.212, j4=-2.938, j5=77.567, j6=-7.639}
  [1231] = {j1=-11.238, j2=59.973, j3=50.534, j4=-2.916, j5=77.364, j6=-7.925}
  [1232] = {j1=-11.245, j2=59.578, j3=50.854, j4=-2.917, j5=77.167, j6=-8.190}
  [1233] = {j1=-11.246, j2=59.187, j3=51.166, j4=-2.941, j5=76.980, j6=-8.431}
  [1234] = {j1=-11.246, j2=59.168, j3=51.187, j4=-2.941, j5=76.962, j6=-8.440}
  [1235] = {j1=-11.247, j2=59.225, j3=51.085, j4=-2.931, j5=77.111, j6=-8.340}
  [1236] = {j1=-11.248, j2=59.233, j3=51.084, j4=-2.928, j5=77.105, j6=-8.333}
  [1237] = {j1=-11.248, j2=59.611, j3=50.795, j4=-2.902, j5=77.263, j6=-8.094}
  [1238] = {j1=-11.242, j2=59.993, j3=50.499, j4=-2.898, j5=77.432, j6=-7.833}
  [1239] = {j1=-11.229, j2=60.376, j3=50.201, j4=-2.918, j5=77.609, j6=-7.549}
  [1240] = {j1=-11.208, j2=60.759, j3=49.904, j4=-2.963, j5=77.788, j6=-7.245}
  [1241] = {j1=-11.182, j2=61.195, j3=49.568, j4=-3.029, j5=77.998, j6=-6.883}
  [1242] = {j1=-11.157, j2=61.629, j3=49.235, j4=-3.090, j5=78.214, j6=-6.519}
  [1243] = {j1=-11.135, j2=62.063, j3=48.901, j4=-3.147, j5=78.439, j6=-6.150}
  [1244] = {j1=-11.115, j2=62.499, j3=48.563, j4=-3.196, j5=78.677, j6=-5.776}
  [1245] = {j1=-11.098, j2=62.940, j3=48.217, j4=-3.238, j5=78.931, j6=-5.395}
  [1246] = {j1=-11.084, j2=63.386, j3=47.859, j4=-3.271, j5=79.206, j6=-5.007}
  [1247] = {j1=-11.073, j2=63.841, j3=47.486, j4=-3.292, j5=79.505, j6=-4.610}
  [1248] = {j1=-11.072, j2=63.916, j3=47.427, j4=-3.295, j5=79.549, j6=-4.540}
  [1249] = {j1=-11.049, j2=64.373, j3=47.047, j4=-3.362, j5=79.861, j6=-4.108}
  [1250] = {j1=-10.998, j2=64.891, j3=46.637, j4=-3.538, j5=80.181, j6=-3.571}
  [1251] = {j1=-10.926, j2=65.355, j3=46.330, j4=-3.814, j5=80.375, j6=-3.054}
  [1252] = {j1=-10.861, j2=65.675, j3=46.189, j4=-4.071, j5=80.394, j6=-2.697}
  [1253] = {j1=-10.802, j2=65.945, j3=46.140, j4=-4.318, j5=80.296, j6=-2.419}
  [1254] = {j1=-10.748, j2=66.171, j3=46.168, j4=-4.559, j5=80.099, j6=-2.207}
  [1255] = {j1=-10.695, j2=66.360, j3=46.258, j4=-4.799, j5=79.820, j6=-2.049}
  [1256] = {j1=-10.644, j2=66.519, j3=46.397, j4=-5.043, j5=79.474, j6=-1.933}
  [1257] = {j1=-10.593, j2=66.654, j3=46.571, j4=-5.294, j5=79.078, j6=-1.848}
  [1258] = {j1=-10.592, j2=66.676, j3=46.534, j4=-5.297, j5=79.151, j6=-1.785}
  [1259] = {j1=-10.644, j2=66.529, j3=46.380, j4=-5.042, j5=79.519, j6=-1.873}
  [1260] = {j1=-10.696, j2=66.358, j3=46.261, j4=-4.795, j5=79.837, j6=-1.991}
  [1261] = {j1=-10.750, j2=66.157, j3=46.192, j4=-4.551, j5=80.089, j6=-2.151}
  [1262] = {j1=-10.806, j2=65.920, j3=46.185, j4=-4.306, j5=80.259, j6=-2.365}
  [1263] = {j1=-10.866, j2=65.639, j3=46.255, j4=-4.055, j5=80.330, j6=-2.645}
  [1264] = {j1=-10.931, j2=65.307, j3=46.415, j4=-3.792, j5=80.287, j6=-3.003}
  [1265] = {j1=-11.005, j2=64.833, j3=46.740, j4=-3.512, j5=80.071, j6=-3.520}
  [1266] = {j1=-11.057, j2=64.306, j3=47.166, j4=-3.332, j5=79.730, j6=-4.055}
  [1267] = {j1=-11.080, j2=63.839, j3=47.565, j4=-3.262, j5=79.396, j6=-4.486}
  [1268] = {j1=-11.083, j2=63.752, j3=47.644, j4=-3.257, j5=79.326, j6=-4.556}
  [1269] = {j1=-11.095, j2=63.286, j3=48.038, j4=-3.233, j5=79.002, j6=-4.953}
  [1270] = {j1=-11.110, j2=62.827, j3=48.418, j4=-3.198, j5=78.701, j6=-5.342}
  [1271] = {j1=-11.128, j2=62.373, j3=48.788, j4=-3.154, j5=78.418, j6=-5.724}
  [1272] = {j1=-11.149, j2=61.923, j3=49.151, j4=-3.101, j5=78.151, j6=-6.100}
  [1273] = {j1=-11.172, j2=61.475, j3=49.509, j4=-3.041, j5=77.897, j6=-6.471}
  [1274] = {j1=-11.198, j2=61.027, j3=49.867, j4=-2.976, j5=77.653, j6=-6.838}
